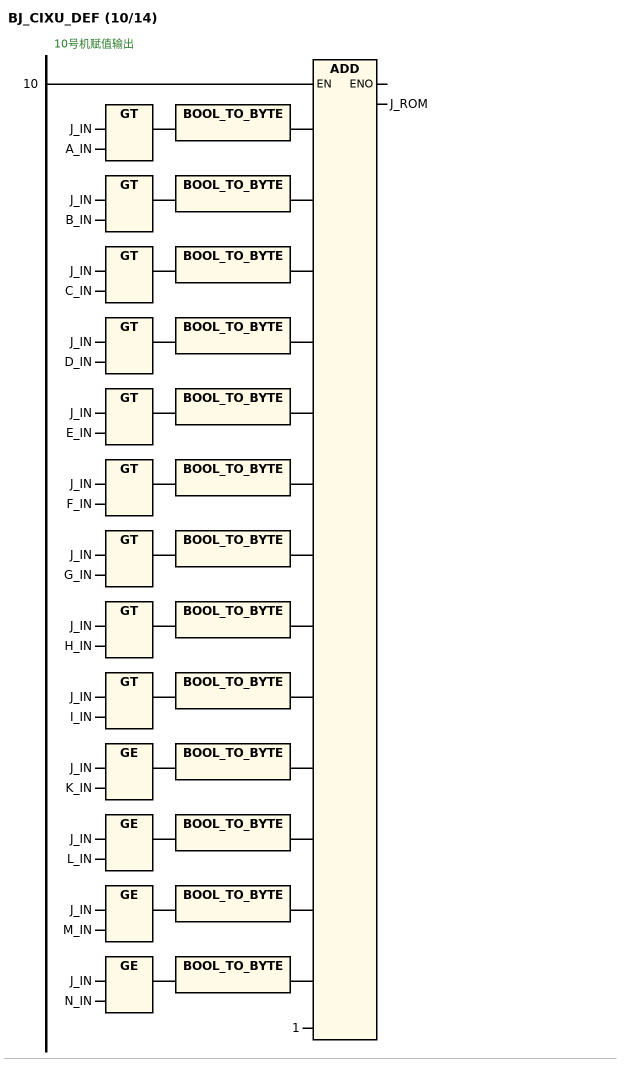
[picture p96: BJ_CIXU_DEF (LD)]
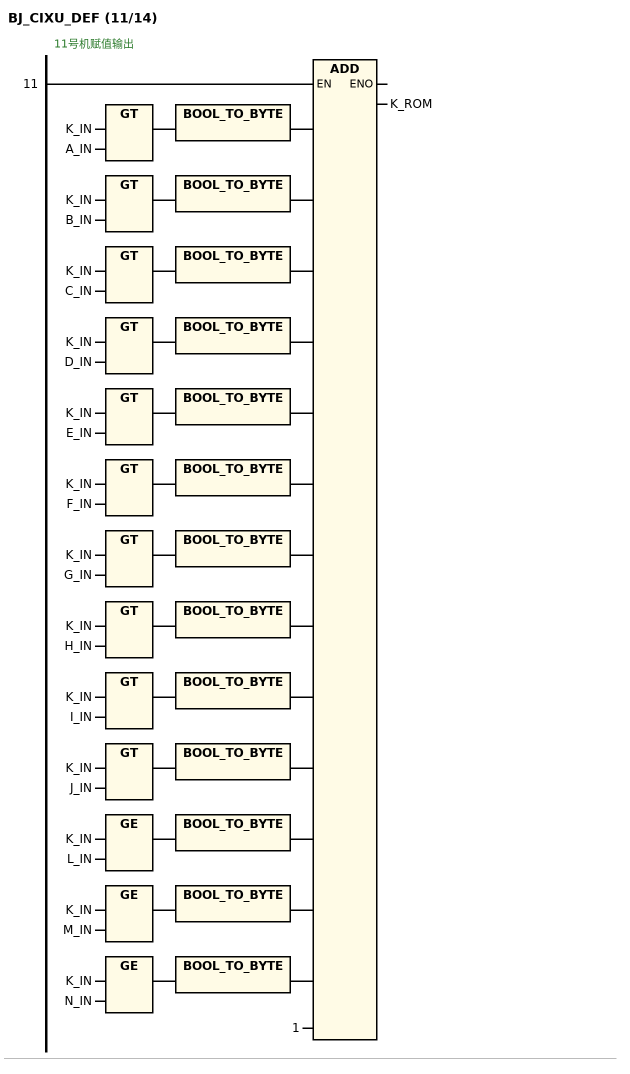
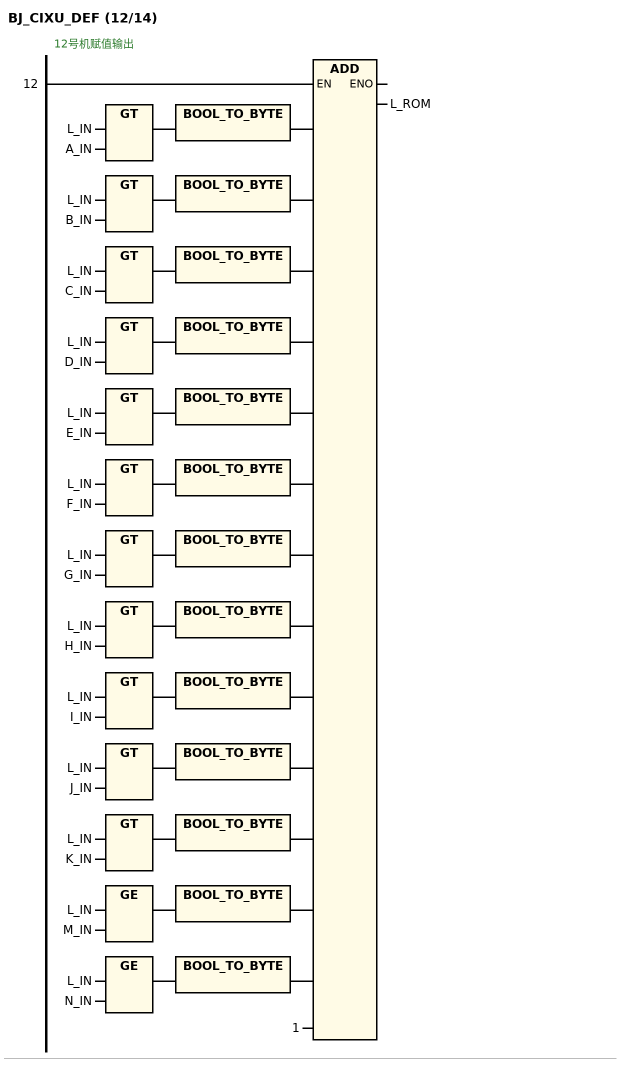
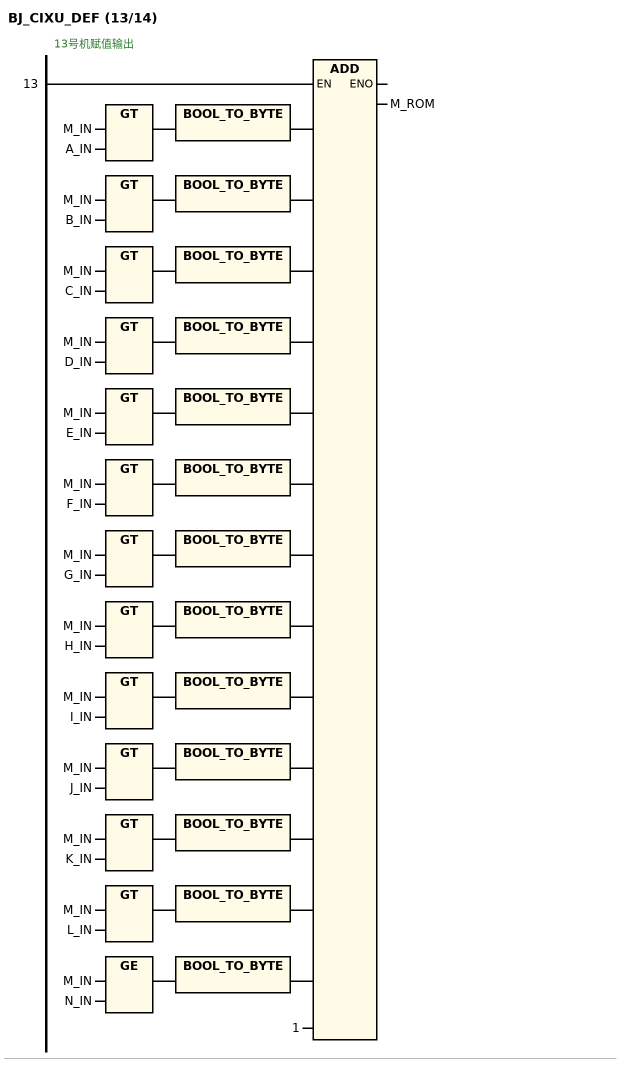
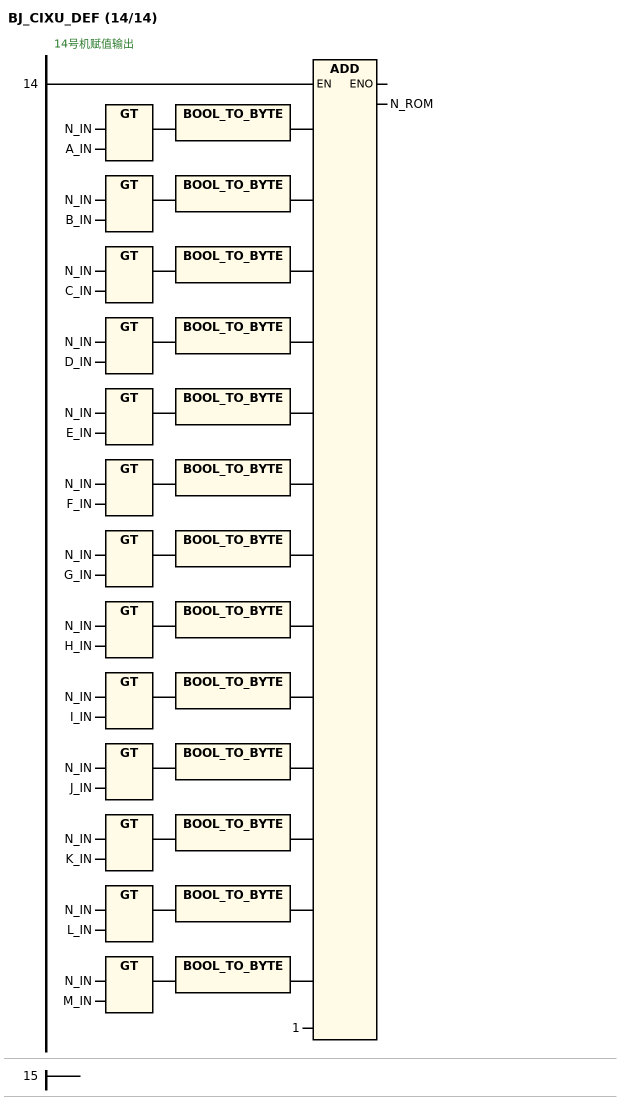
_LD_ (* Ladder Diagram *)
NETWORK 1 (* 1号机赋值输出 *)
	*
		EN --- ADD(BOOL_TO_BYTE(GE(A_IN, B_IN)), BOOL_TO_BYTE(GE(A_IN, C_IN)), BOOL_TO_BYTE(GE(A_IN, D_IN)), BOOL_TO_BYTE(GE(A_IN, E_IN)), BOOL_TO_BYTE(GE(A_IN, F_IN)), BOOL_TO_BYTE(GE(A_IN, G_IN)), BOOL_TO_BYTE(GE(A_IN, H_IN)), BOOL_TO_BYTE(GE(A_IN, I_IN)), BOOL_TO_BYTE(GE(A_IN, J_IN)), BOOL_TO_BYTE(GE(A_IN, K_IN)), BOOL_TO_BYTE(GE(A_IN, L_IN)), BOOL_TO_BYTE(GE(A_IN, M_IN)), BOOL_TO_BYTE(GE(A_IN, N_IN)), 1) => A_ROM
NETWORK 2 (* 2号机赋值输出 *)
	*
		EN --- ADD(BOOL_TO_BYTE(GT(B_IN, A_IN)), BOOL_TO_BYTE(GE(B_IN, C_IN)), BOOL_TO_BYTE(GE(B_IN, D_IN)), BOOL_TO_BYTE(GE(B_IN, E_IN)), BOOL_TO_BYTE(GE(B_IN, F_IN)), BOOL_TO_BYTE(GE(B_IN, G_IN)), BOOL_TO_BYTE(GE(B_IN, H_IN)), BOOL_TO_BYTE(GE(B_IN, I_IN)), BOOL_TO_BYTE(GE(B_IN, J_IN)), BOOL_TO_BYTE(GE(B_IN, K_IN)), BOOL_TO_BYTE(GE(B_IN, L_IN)), BOOL_TO_BYTE(GE(B_IN, M_IN)), BOOL_TO_BYTE(GE(B_IN, N_IN)), 1) => B_ROM
NETWORK 3 (* 3号机赋值输出 *)
	*
		EN --- ADD(BOOL_TO_BYTE(GT(C_IN, A_IN)), BOOL_TO_BYTE(GT(C_IN, B_IN)), BOOL_TO_BYTE(GE(C_IN, D_IN)), BOOL_TO_BYTE(GE(C_IN, E_IN)), BOOL_TO_BYTE(GE(C_IN, F_IN)), BOOL_TO_BYTE(GE(C_IN, G_IN)), BOOL_TO_BYTE(GE(C_IN, H_IN)), BOOL_TO_BYTE(GE(C_IN, I_IN)), BOOL_TO_BYTE(GE(C_IN, J_IN)), BOOL_TO_BYTE(GE(C_IN, K_IN)), BOOL_TO_BYTE(GE(C_IN, L_IN)), BOOL_TO_BYTE(GE(C_IN, M_IN)), BOOL_TO_BYTE(GE(C_IN, N_IN)), 1) => C_ROM
NETWORK 4 (* 4号机赋值输出 *)
	*
		EN --- ADD(BOOL_TO_BYTE(GT(D_IN, A_IN)), BOOL_TO_BYTE(GT(D_IN, B_IN)), BOOL_TO_BYTE(GT(D_IN, C_IN)), BOOL_TO_BYTE(GE(D_IN, E_IN)), BOOL_TO_BYTE(GE(D_IN, F_IN)), BOOL_TO_BYTE(GE(D_IN, G_IN)), BOOL_TO_BYTE(GE(D_IN, H_IN)), BOOL_TO_BYTE(GE(D_IN, I_IN)), BOOL_TO_BYTE(GE(D_IN, J_IN)), BOOL_TO_BYTE(GE(D_IN, K_IN)), BOOL_TO_BYTE(GE(D_IN, L_IN)), BOOL_TO_BYTE(GE(D_IN, M_IN)), BOOL_TO_BYTE(GE(D_IN, N_IN)), 1) => D_ROM
NETWORK 5 (* 5号机赋值输出 *)
	*
		EN --- ADD(BOOL_TO_BYTE(GT(E_IN, A_IN)), BOOL_TO_BYTE(GT(E_IN, B_IN)), BOOL_TO_BYTE(GT(E_IN, C_IN)), BOOL_TO_BYTE(GT(E_IN, D_IN)), BOOL_TO_BYTE(GE(E_IN, F_IN)), BOOL_TO_BYTE(GE(E_IN, G_IN)), BOOL_TO_BYTE(GE(E_IN, H_IN)), BOOL_TO_BYTE(GE(E_IN, I_IN)), BOOL_TO_BYTE(GE(E_IN, J_IN)), BOOL_TO_BYTE(GE(E_IN, K_IN)), BOOL_TO_BYTE(GE(E_IN, L_IN)), BOOL_TO_BYTE(GE(E_IN, M_IN)), BOOL_TO_BYTE(GE(E_IN, N_IN)), 1) => E_ROM
NETWORK 6 (* 6号机赋值输出 *)
	*
		EN --- ADD(BOOL_TO_BYTE(GT(F_IN, A_IN)), BOOL_TO_BYTE(GT(F_IN, B_IN)), BOOL_TO_BYTE(GT(F_IN, C_IN)), BOOL_TO_BYTE(GT(F_IN, D_IN)), BOOL_TO_BYTE(GT(F_IN, E_IN)), BOOL_TO_BYTE(GE(F_IN, G_IN)), BOOL_TO_BYTE(GE(F_IN, H_IN)), BOOL_TO_BYTE(GE(F_IN, I_IN)), BOOL_TO_BYTE(GE(F_IN, J_IN)), BOOL_TO_BYTE(GE(F_IN, K_IN)), BOOL_TO_BYTE(GE(F_IN, L_IN)), BOOL_TO_BYTE(GE(F_IN, M_IN)), BOOL_TO_BYTE(GE(F_IN, N_IN)), 1) => F_ROM
NETWORK 7 (* 7号机赋值输出 *)
	*
		EN --- ADD(BOOL_TO_BYTE(GT(G_IN, A_IN)), BOOL_TO_BYTE(GT(G_IN, B_IN)), BOOL_TO_BYTE(GT(G_IN, C_IN)), BOOL_TO_BYTE(GT(G_IN, D_IN)), BOOL_TO_BYTE(GT(G_IN, E_IN)), BOOL_TO_BYTE(GT(G_IN, F_IN)), BOOL_TO_BYTE(GE(G_IN, H_IN)), BOOL_TO_BYTE(GE(G_IN, I_IN)), BOOL_TO_BYTE(GE(G_IN, J_IN)), BOOL_TO_BYTE(GE(G_IN, K_IN)), BOOL_TO_BYTE(GE(G_IN, L_IN)), BOOL_TO_BYTE(GE(G_IN, M_IN)), BOOL_TO_BYTE(GE(G_IN, N_IN)), 1) => G_ROM
NETWORK 8 (* 8号机赋值输出 *)
	*
		EN --- ADD(BOOL_TO_BYTE(GT(H_IN, A_IN)), BOOL_TO_BYTE(GT(H_IN, B_IN)), BOOL_TO_BYTE(GT(H_IN, C_IN)), BOOL_TO_BYTE(GT(H_IN, D_IN)), BOOL_TO_BYTE(GT(H_IN, E_IN)), BOOL_TO_BYTE(GT(H_IN, F_IN)), BOOL_TO_BYTE(GT(H_IN, G_IN)), BOOL_TO_BYTE(GE(H_IN, I_IN)), BOOL_TO_BYTE(GE(H_IN, J_IN)), BOOL_TO_BYTE(GE(H_IN, K_IN)), BOOL_TO_BYTE(GE(H_IN, L_IN)), BOOL_TO_BYTE(GE(H_IN, M_IN)), BOOL_TO_BYTE(GE(H_IN, N_IN)), 1) => H_ROM
NETWORK 9 (* 9号机赋值输出 *)
	*
		EN --- ADD(BOOL_TO_BYTE(GT(I_IN, A_IN)), BOOL_TO_BYTE(GT(I_IN, B_IN)), BOOL_TO_BYTE(GT(I_IN, C_IN)), BOOL_TO_BYTE(GT(I_IN, D_IN)), BOOL_TO_BYTE(GT(I_IN, E_IN)), BOOL_TO_BYTE(GT(I_IN, F_IN)), BOOL_TO_BYTE(GT(I_IN, G_IN)), BOOL_TO_BYTE(GT(I_IN, H_IN)), BOOL_TO_BYTE(GE(I_IN, J_IN)), BOOL_TO_BYTE(GE(I_IN, K_IN)), BOOL_TO_BYTE(GE(I_IN, L_IN)), BOOL_TO_BYTE(GE(I_IN, M_IN)), BOOL_TO_BYTE(GE(I_IN, N_IN)), 1) => I_ROM
NETWORK 10 (* 10号机赋值输出 *)
	*
		EN --- ADD(BOOL_TO_BYTE(GT(J_IN, A_IN)), BOOL_TO_BYTE(GT(J_IN, B_IN)), BOOL_TO_BYTE(GT(J_IN, C_IN)), BOOL_TO_BYTE(GT(J_IN, D_IN)), BOOL_TO_BYTE(GT(J_IN, E_IN)), BOOL_TO_BYTE(GT(J_IN, F_IN)), BOOL_TO_BYTE(GT(J_IN, G_IN)), BOOL_TO_BYTE(GT(J_IN, H_IN)), BOOL_TO_BYTE(GT(J_IN, I_IN)), BOOL_TO_BYTE(GE(J_IN, K_IN)), BOOL_TO_BYTE(GE(J_IN, L_IN)), BOOL_TO_BYTE(GE(J_IN, M_IN)), BOOL_TO_BYTE(GE(J_IN, N_IN)), 1) => J_ROM
NETWORK 11 (* 11号机赋值输出 *)
	*
		EN --- ADD(BOOL_TO_BYTE(GT(K_IN, A_IN)), BOOL_TO_BYTE(GT(K_IN, B_IN)), BOOL_TO_BYTE(GT(K_IN, C_IN)), BOOL_TO_BYTE(GT(K_IN, D_IN)), BOOL_TO_BYTE(GT(K_IN, E_IN)), BOOL_TO_BYTE(GT(K_IN, F_IN)), BOOL_TO_BYTE(GT(K_IN, G_IN)), BOOL_TO_BYTE(GT(K_IN, H_IN)), BOOL_TO_BYTE(GT(K_IN, I_IN)), BOOL_TO_BYTE(GT(K_IN, J_IN)), BOOL_TO_BYTE(GE(K_IN, L_IN)), BOOL_TO_BYTE(GE(K_IN, M_IN)), BOOL_TO_BYTE(GE(K_IN, N_IN)), 1) => K_ROM
NETWORK 12 (* 12号机赋值输出 *)
	*
		EN --- ADD(BOOL_TO_BYTE(GT(L_IN, A_IN)), BOOL_TO_BYTE(GT(L_IN, B_IN)), BOOL_TO_BYTE(GT(L_IN, C_IN)), BOOL_TO_BYTE(GT(L_IN, D_IN)), BOOL_TO_BYTE(GT(L_IN, E_IN)), BOOL_TO_BYTE(GT(L_IN, F_IN)), BOOL_TO_BYTE(GT(L_IN, G_IN)), BOOL_TO_BYTE(GT(L_IN, H_IN)), BOOL_TO_BYTE(GT(L_IN, I_IN)), BOOL_TO_BYTE(GT(L_IN, J_IN)), BOOL_TO_BYTE(GT(L_IN, K_IN)), BOOL_TO_BYTE(GE(L_IN, M_IN)), BOOL_TO_BYTE(GE(L_IN, N_IN)), 1) => L_ROM
NETWORK 13 (* 13号机赋值输出 *)
	*
		EN --- ADD(BOOL_TO_BYTE(GT(M_IN, A_IN)), BOOL_TO_BYTE(GT(M_IN, B_IN)), BOOL_TO_BYTE(GT(M_IN, C_IN)), BOOL_TO_BYTE(GT(M_IN, D_IN)), BOOL_TO_BYTE(GT(M_IN, E_IN)), BOOL_TO_BYTE(GT(M_IN, F_IN)), BOOL_TO_BYTE(GT(M_IN, G_IN)), BOOL_TO_BYTE(GT(M_IN, H_IN)), BOOL_TO_BYTE(GT(M_IN, I_IN)), BOOL_TO_BYTE(GT(M_IN, J_IN)), BOOL_TO_BYTE(GT(M_IN, K_IN)), BOOL_TO_BYTE(GT(M_IN, L_IN)), BOOL_TO_BYTE(GE(M_IN, N_IN)), 1) => M_ROM
NETWORK 14 (* 14号机赋值输出 *)
	*
		EN --- ADD(BOOL_TO_BYTE(GT(N_IN, A_IN)), BOOL_TO_BYTE(GT(N_IN, B_IN)), BOOL_TO_BYTE(GT(N_IN, C_IN)), BOOL_TO_BYTE(GT(N_IN, D_IN)), BOOL_TO_BYTE(GT(N_IN, E_IN)), BOOL_TO_BYTE(GT(N_IN, F_IN)), BOOL_TO_BYTE(GT(N_IN, G_IN)), BOOL_TO_BYTE(GT(N_IN, H_IN)), BOOL_TO_BYTE(GT(N_IN, I_IN)), BOOL_TO_BYTE(GT(N_IN, J_IN)), BOOL_TO_BYTE(GT(N_IN, K_IN)), BOOL_TO_BYTE(GT(N_IN, L_IN)), BOOL_TO_BYTE(GT(N_IN, M_IN)), 1) => N_ROM
NETWORK 15
	*
_END_LD_
(* the same logic as Structured Text *)
(* Network 1: 1号机赋值输出 *)
A_ROM := BOOL_TO_BYTE(A_IN >= B_IN) + BOOL_TO_BYTE(A_IN >= C_IN) + BOOL_TO_BYTE(A_IN >= D_IN) + BOOL_TO_BYTE(A_IN >= E_IN) + BOOL_TO_BYTE(A_IN >= F_IN) + BOOL_TO_BYTE(A_IN >= G_IN) + BOOL_TO_BYTE(A_IN >= H_IN) + BOOL_TO_BYTE(A_IN >= I_IN) + BOOL_TO_BYTE(A_IN >= J_IN) + BOOL_TO_BYTE(A_IN >= K_IN) + BOOL_TO_BYTE(A_IN >= L_IN) + BOOL_TO_BYTE(A_IN >= M_IN) + BOOL_TO_BYTE(A_IN >= N_IN) + 1;
(* Network 2: 2号机赋值输出 *)
B_ROM := BOOL_TO_BYTE(B_IN > A_IN) + BOOL_TO_BYTE(B_IN >= C_IN) + BOOL_TO_BYTE(B_IN >= D_IN) + BOOL_TO_BYTE(B_IN >= E_IN) + BOOL_TO_BYTE(B_IN >= F_IN) + BOOL_TO_BYTE(B_IN >= G_IN) + BOOL_TO_BYTE(B_IN >= H_IN) + BOOL_TO_BYTE(B_IN >= I_IN) + BOOL_TO_BYTE(B_IN >= J_IN) + BOOL_TO_BYTE(B_IN >= K_IN) + BOOL_TO_BYTE(B_IN >= L_IN) + BOOL_TO_BYTE(B_IN >= M_IN) + BOOL_TO_BYTE(B_IN >= N_IN) + 1;
(* Network 3: 3号机赋值输出 *)
C_ROM := BOOL_TO_BYTE(C_IN > A_IN) + BOOL_TO_BYTE(C_IN > B_IN) + BOOL_TO_BYTE(C_IN >= D_IN) + BOOL_TO_BYTE(C_IN >= E_IN) + BOOL_TO_BYTE(C_IN >= F_IN) + BOOL_TO_BYTE(C_IN >= G_IN) + BOOL_TO_BYTE(C_IN >= H_IN) + BOOL_TO_BYTE(C_IN >= I_IN) + BOOL_TO_BYTE(C_IN >= J_IN) + BOOL_TO_BYTE(C_IN >= K_IN) + BOOL_TO_BYTE(C_IN >= L_IN) + BOOL_TO_BYTE(C_IN >= M_IN) + BOOL_TO_BYTE(C_IN >= N_IN) + 1;
(* Network 4: 4号机赋值输出 *)
D_ROM := BOOL_TO_BYTE(D_IN > A_IN) + BOOL_TO_BYTE(D_IN > B_IN) + BOOL_TO_BYTE(D_IN > C_IN) + BOOL_TO_BYTE(D_IN >= E_IN) + BOOL_TO_BYTE(D_IN >= F_IN) + BOOL_TO_BYTE(D_IN >= G_IN) + BOOL_TO_BYTE(D_IN >= H_IN) + BOOL_TO_BYTE(D_IN >= I_IN) + BOOL_TO_BYTE(D_IN >= J_IN) + BOOL_TO_BYTE(D_IN >= K_IN) + BOOL_TO_BYTE(D_IN >= L_IN) + BOOL_TO_BYTE(D_IN >= M_IN) + BOOL_TO_BYTE(D_IN >= N_IN) + 1;
(* Network 5: 5号机赋值输出 *)
E_ROM := BOOL_TO_BYTE(E_IN > A_IN) + BOOL_TO_BYTE(E_IN > B_IN) + BOOL_TO_BYTE(E_IN > C_IN) + BOOL_TO_BYTE(E_IN > D_IN) + BOOL_TO_BYTE(E_IN >= F_IN) + BOOL_TO_BYTE(E_IN >= G_IN) + BOOL_TO_BYTE(E_IN >= H_IN) + BOOL_TO_BYTE(E_IN >= I_IN) + BOOL_TO_BYTE(E_IN >= J_IN) + BOOL_TO_BYTE(E_IN >= K_IN) + BOOL_TO_BYTE(E_IN >= L_IN) + BOOL_TO_BYTE(E_IN >= M_IN) + BOOL_TO_BYTE(E_IN >= N_IN) + 1;
(* Network 6: 6号机赋值输出 *)
F_ROM := BOOL_TO_BYTE(F_IN > A_IN) + BOOL_TO_BYTE(F_IN > B_IN) + BOOL_TO_BYTE(F_IN > C_IN) + BOOL_TO_BYTE(F_IN > D_IN) + BOOL_TO_BYTE(F_IN > E_IN) + BOOL_TO_BYTE(F_IN >= G_IN) + BOOL_TO_BYTE(F_IN >= H_IN) + BOOL_TO_BYTE(F_IN >= I_IN) + BOOL_TO_BYTE(F_IN >= J_IN) + BOOL_TO_BYTE(F_IN >= K_IN) + BOOL_TO_BYTE(F_IN >= L_IN) + BOOL_TO_BYTE(F_IN >= M_IN) + BOOL_TO_BYTE(F_IN >= N_IN) + 1;
(* Network 7: 7号机赋值输出 *)
G_ROM := BOOL_TO_BYTE(G_IN > A_IN) + BOOL_TO_BYTE(G_IN > B_IN) + BOOL_TO_BYTE(G_IN > C_IN) + BOOL_TO_BYTE(G_IN > D_IN) + BOOL_TO_BYTE(G_IN > E_IN) + BOOL_TO_BYTE(G_IN > F_IN) + BOOL_TO_BYTE(G_IN >= H_IN) + BOOL_TO_BYTE(G_IN >= I_IN) + BOOL_TO_BYTE(G_IN >= J_IN) + BOOL_TO_BYTE(G_IN >= K_IN) + BOOL_TO_BYTE(G_IN >= L_IN) + BOOL_TO_BYTE(G_IN >= M_IN) + BOOL_TO_BYTE(G_IN >= N_IN) + 1;
(* Network 8: 8号机赋值输出 *)
H_ROM := BOOL_TO_BYTE(H_IN > A_IN) + BOOL_TO_BYTE(H_IN > B_IN) + BOOL_TO_BYTE(H_IN > C_IN) + BOOL_TO_BYTE(H_IN > D_IN) + BOOL_TO_BYTE(H_IN > E_IN) + BOOL_TO_BYTE(H_IN > F_IN) + BOOL_TO_BYTE(H_IN > G_IN) + BOOL_TO_BYTE(H_IN >= I_IN) + BOOL_TO_BYTE(H_IN >= J_IN) + BOOL_TO_BYTE(H_IN >= K_IN) + BOOL_TO_BYTE(H_IN >= L_IN) + BOOL_TO_BYTE(H_IN >= M_IN) + BOOL_TO_BYTE(H_IN >= N_IN) + 1;
(* Network 9: 9号机赋值输出 *)
I_ROM := BOOL_TO_BYTE(I_IN > A_IN) + BOOL_TO_BYTE(I_IN > B_IN) + BOOL_TO_BYTE(I_IN > C_IN) + BOOL_TO_BYTE(I_IN > D_IN) + BOOL_TO_BYTE(I_IN > E_IN) + BOOL_TO_BYTE(I_IN > F_IN) + BOOL_TO_BYTE(I_IN > G_IN) + BOOL_TO_BYTE(I_IN > H_IN) + BOOL_TO_BYTE(I_IN >= J_IN) + BOOL_TO_BYTE(I_IN >= K_IN) + BOOL_TO_BYTE(I_IN >= L_IN) + BOOL_TO_BYTE(I_IN >= M_IN) + BOOL_TO_BYTE(I_IN >= N_IN) + 1;
(* Network 10: 10号机赋值输出 *)
J_ROM := BOOL_TO_BYTE(J_IN > A_IN) + BOOL_TO_BYTE(J_IN > B_IN) + BOOL_TO_BYTE(J_IN > C_IN) + BOOL_TO_BYTE(J_IN > D_IN) + BOOL_TO_BYTE(J_IN > E_IN) + BOOL_TO_BYTE(J_IN > F_IN) + BOOL_TO_BYTE(J_IN > G_IN) + BOOL_TO_BYTE(J_IN > H_IN) + BOOL_TO_BYTE(J_IN > I_IN) + BOOL_TO_BYTE(J_IN >= K_IN) + BOOL_TO_BYTE(J_IN >= L_IN) + BOOL_TO_BYTE(J_IN >= M_IN) + BOOL_TO_BYTE(J_IN >= N_IN) + 1;
(* Network 11: 11号机赋值输出 *)
K_ROM := BOOL_TO_BYTE(K_IN > A_IN) + BOOL_TO_BYTE(K_IN > B_IN) + BOOL_TO_BYTE(K_IN > C_IN) + BOOL_TO_BYTE(K_IN > D_IN) + BOOL_TO_BYTE(K_IN > E_IN) + BOOL_TO_BYTE(K_IN > F_IN) + BOOL_TO_BYTE(K_IN > G_IN) + BOOL_TO_BYTE(K_IN > H_IN) + BOOL_TO_BYTE(K_IN > I_IN) + BOOL_TO_BYTE(K_IN > J_IN) + BOOL_TO_BYTE(K_IN >= L_IN) + BOOL_TO_BYTE(K_IN >= M_IN) + BOOL_TO_BYTE(K_IN >= N_IN) + 1;
(* Network 12: 12号机赋值输出 *)
L_ROM := BOOL_TO_BYTE(L_IN > A_IN) + BOOL_TO_BYTE(L_IN > B_IN) + BOOL_TO_BYTE(L_IN > C_IN) + BOOL_TO_BYTE(L_IN > D_IN) + BOOL_TO_BYTE(L_IN > E_IN) + BOOL_TO_BYTE(L_IN > F_IN) + BOOL_TO_BYTE(L_IN > G_IN) + BOOL_TO_BYTE(L_IN > H_IN) + BOOL_TO_BYTE(L_IN > I_IN) + BOOL_TO_BYTE(L_IN > J_IN) + BOOL_TO_BYTE(L_IN > K_IN) + BOOL_TO_BYTE(L_IN >= M_IN) + BOOL_TO_BYTE(L_IN >= N_IN) + 1;
(* Network 13: 13号机赋值输出 *)
M_ROM := BOOL_TO_BYTE(M_IN > A_IN) + BOOL_TO_BYTE(M_IN > B_IN) + BOOL_TO_BYTE(M_IN > C_IN) + BOOL_TO_BYTE(M_IN > D_IN) + BOOL_TO_BYTE(M_IN > E_IN) + BOOL_TO_BYTE(M_IN > F_IN) + BOOL_TO_BYTE(M_IN > G_IN) + BOOL_TO_BYTE(M_IN > H_IN) + BOOL_TO_BYTE(M_IN > I_IN) + BOOL_TO_BYTE(M_IN > J_IN) + BOOL_TO_BYTE(M_IN > K_IN) + BOOL_TO_BYTE(M_IN > L_IN) + BOOL_TO_BYTE(M_IN >= N_IN) + 1;
(* Network 14: 14号机赋值输出 *)
N_ROM := BOOL_TO_BYTE(N_IN > A_IN) + BOOL_TO_BYTE(N_IN > B_IN) + BOOL_TO_BYTE(N_IN > C_IN) + BOOL_TO_BYTE(N_IN > D_IN) + BOOL_TO_BYTE(N_IN > E_IN) + BOOL_TO_BYTE(N_IN > F_IN) + BOOL_TO_BYTE(N_IN > G_IN) + BOOL_TO_BYTE(N_IN > H_IN) + BOOL_TO_BYTE(N_IN > I_IN) + BOOL_TO_BYTE(N_IN > J_IN) + BOOL_TO_BYTE(N_IN > K_IN) + BOOL_TO_BYTE(N_IN > L_IN) + BOOL_TO_BYTE(N_IN > M_IN) + 1;
(* Network 15 *)
END_FUNCTION_BLOCK

(* POU DEF_PAIXU, LD *)
FUNCTION_BLOCK DEF_PAIXU
VAR_INPUT
	A_IN: BOOL;
	A_ROM: BYTE;
	B_IN: BOOL;
	B_ROM: BYTE;
	C_IN: BOOL;
	C_ROM: BYTE;
	D_IN: BOOL;
	D_ROM: BYTE;
	E_IN: BOOL;
	E_ROM: BYTE;
	F_IN: BOOL;
	F_ROM: BYTE;
	G_IN: BOOL;
	G_ROM: BYTE;
	H_IN: BOOL;
	H_ROM: BYTE;
	I_IN: BOOL;
	I_ROM: BYTE;
	J_IN: BOOL;
	J_ROM: BYTE;
	K_IN: BOOL;
	K_ROM: BYTE;
	L_IN: BOOL;
	L_ROM: BYTE;
	M_IN: BOOL;
	M_ROM: BYTE;
	N_IN: BOOL;
	N_ROM: BYTE;
	ROM_SHU: WORD;
	PSH_IN: BOOL;
END_VAR
VAR_OUTPUT
	A_DZ: BOOL;
	B_DZ: BOOL;
	C_DZ: BOOL;
	D_DZ: BOOL;
	E_DZ: BOOL;
	F_DZ: BOOL;
	G_DZ: BOOL;
	H_DZ: BOOL;
	I_DZ: BOOL;
	J_DZ: BOOL;
	K_DZ: BOOL;
	L_DZ: BOOL;
	M_DZ: BOOL;
	N_DZ: BOOL;
	A_KA: BOOL;
	B_KA: BOOL;
	C_KA: BOOL;
	D_KA: BOOL;
	E_KA: BOOL;
	F_KA: BOOL;
	G_KA: BOOL;
	H_KA: BOOL;
	  I_KA: BOOL;
	J_KA: BOOL;
	K_KA: BOOL;
	L_KA: BOOL;
       M_KA: BOOL;
	N_KA: BOOL;
	FJ_ROM: BYTE;
	ROM: BYTE;
END_VAR
VAR
	INPUT_KA: BOOL;
	A_0: BOOL;
	B_0: BOOL;
	C_0: BOOL;
	D_0: BOOL;
	F_0: BOOL;
	E_0: BOOL;
	G_0: BOOL;
	H_0: BOOL;

	A_FJ: BOOL;
	B_FJ: BOOL;
	C_FJ: BOOL;
	D_FJ: BOOL;
	E_FJ: BOOL;
	F_FJ: BOOL;
	G_FJ: BOOL;
	H_FJ: BOOL;
	I_0: BOOL;

	J_FJ: BOOL;
	J_0: BOOL;
	I_FJ: BOOL;
	KA_FJ: BOOL;
	ROM_1: BOOL;
	ROM_2: BOOL;
	ROM_3: BOOL;
	ROM_4: BOOL;
	ROM_10: BOOL;
	ROM_9: BOOL;
	ROM_8: BOOL;
	ROM_7: BOOL;
	ROM_6: BOOL;
	ROM_5: BOOL;
	FJ_CTU: CTU;
	CTU_Q: BOOL;
	CV: WORD;
	CV_0: BOOL;
	CV_1: BOOL;
	CV_2: BOOL;
	CV_3: BOOL;
	CV_4: BOOL;
	CV_5: BOOL;
	CV_6: BOOL;
	CV_7: BOOL;
	CV_8: BOOL;
	CV_9: BOOL;
	KAIKU_SHU: WORD;
	ROM_0: BOOL;
	KU_SHU: WORD;
	ROM_11: BOOL;
	ROM_12: BOOL;
	ROM_13: BOOL;
	ROM_14: BOOL;
	K_0: BOOL;
	K_FJ: BOOL;
	L_0: BOOL;
	L_FJ: BOOL;
	M_0: BOOL;
	M_FJ: BOOL;
	N_0: BOOL;
	N_FJ: BOOL;
	CV_10: BOOL;
	CV_11: BOOL;
	CV_12: BOOL;
	CV_13: BOOL;
	A_15: BOOL;
	B_15: BOOL;
	C_15: BOOL;
	D_15: BOOL;
	E_15: BOOL;
	F_15: BOOL;
	H_15: BOOL;
	I_15: BOOL;
	J_15: BOOL;
	K_15: BOOL;
	L_15: BOOL;
	M_15: BOOL;
	N_15: BOOL;
	G_15: BOOL;
END_VAR
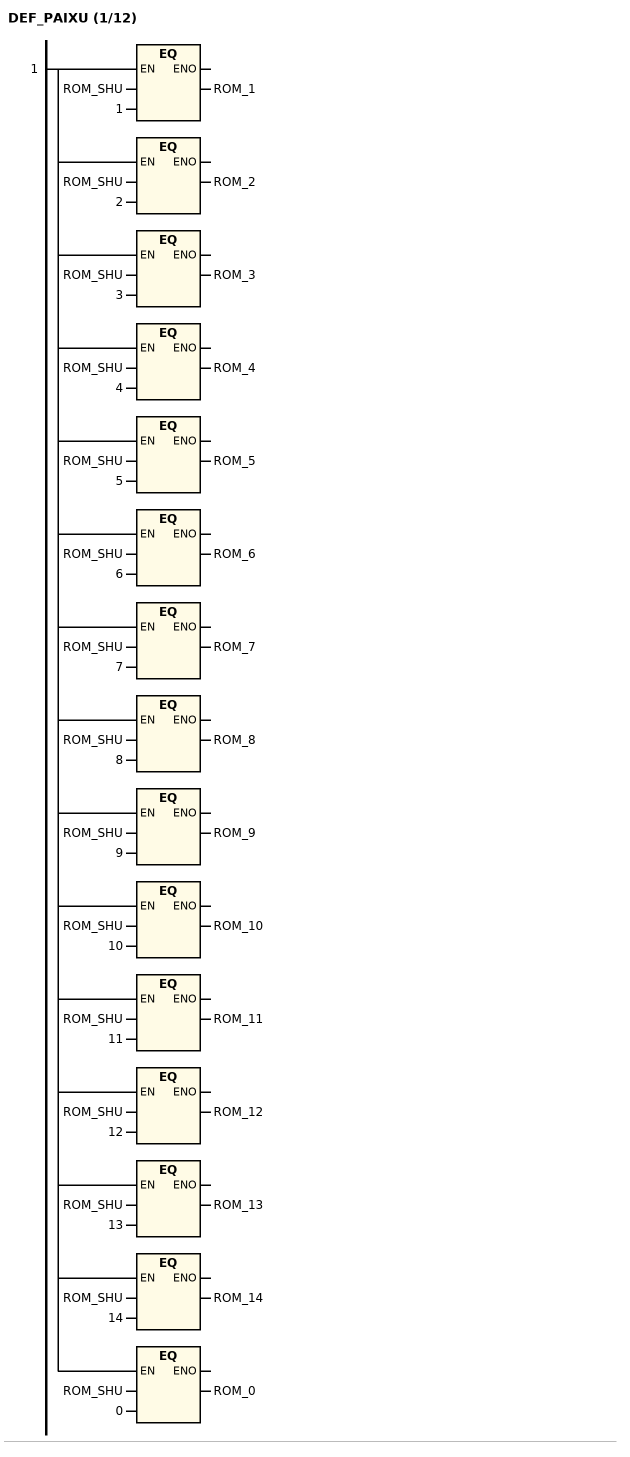
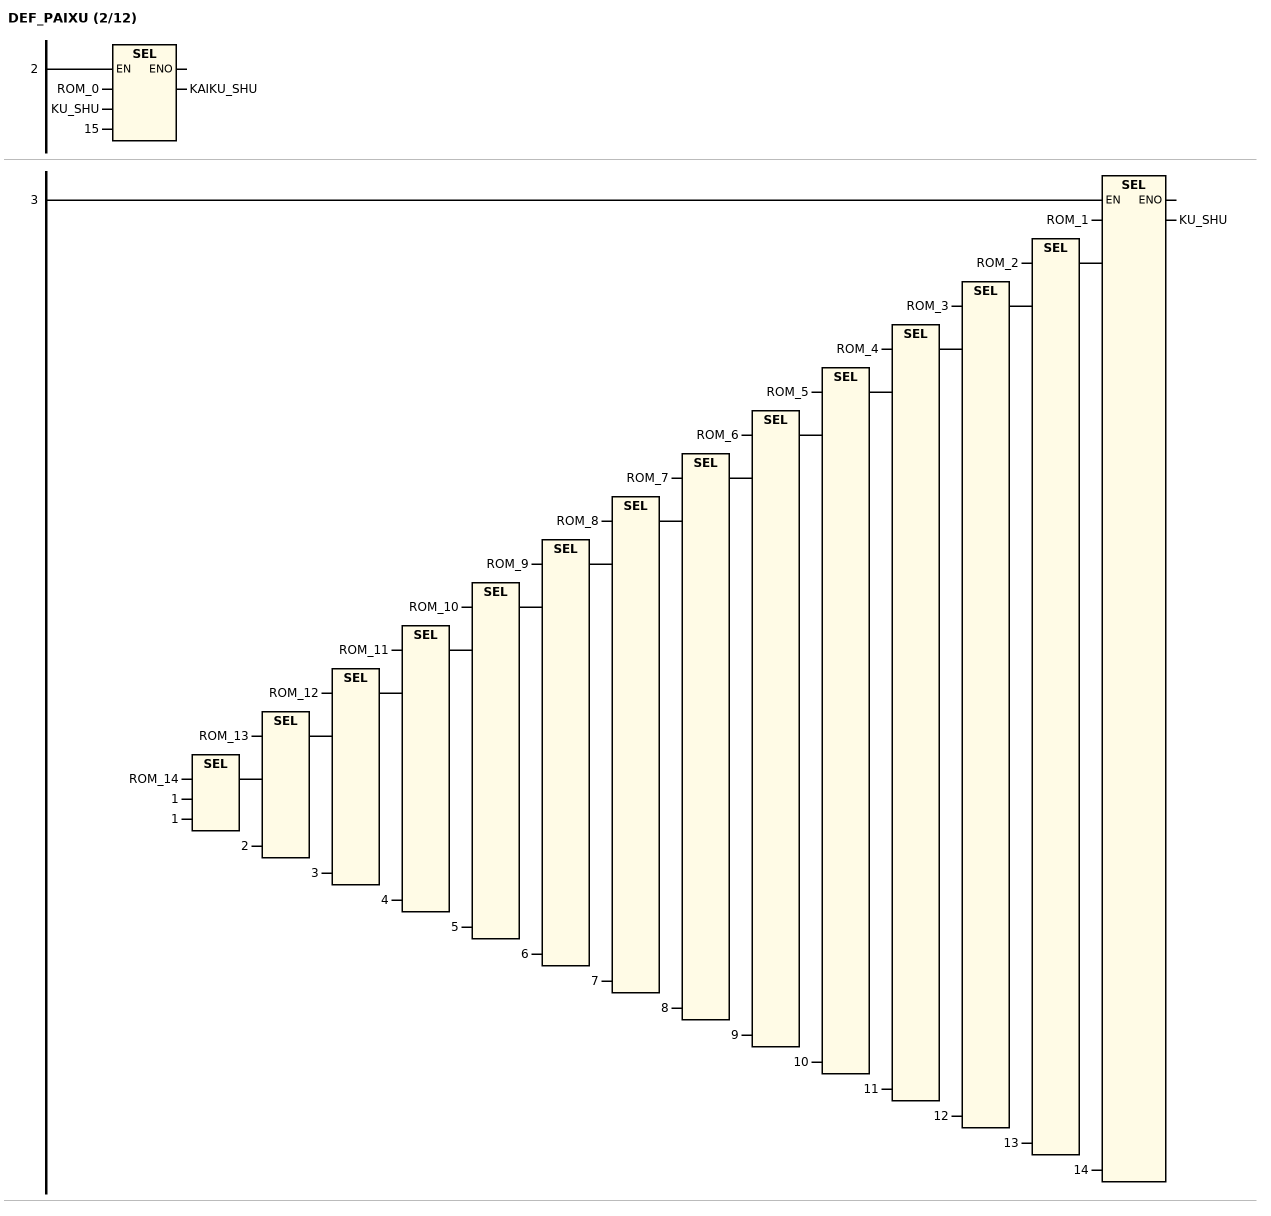
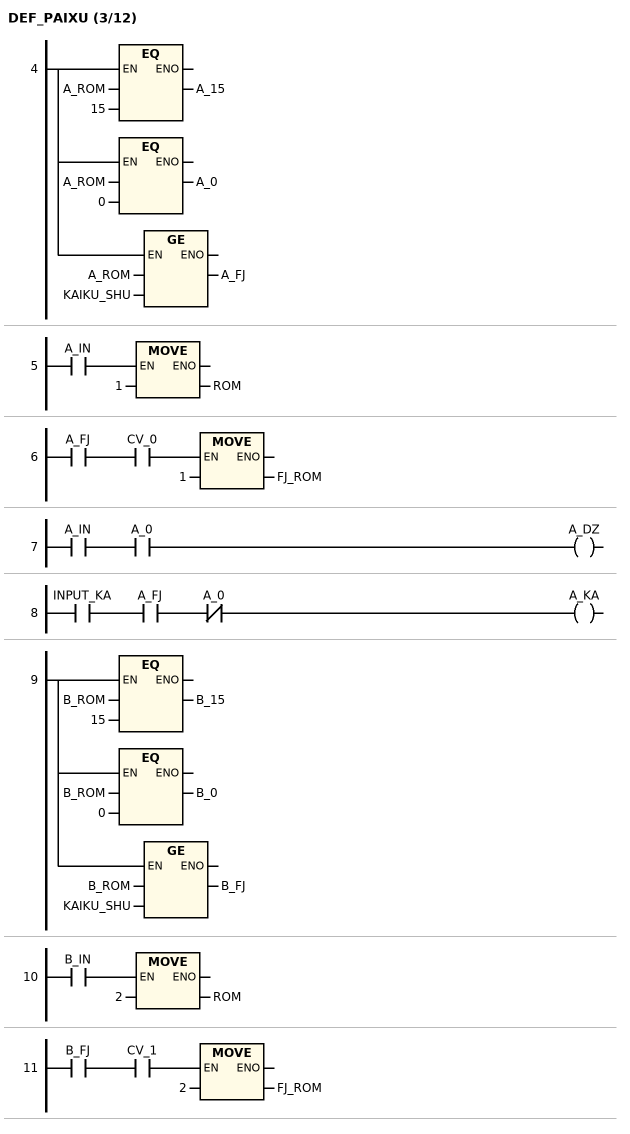
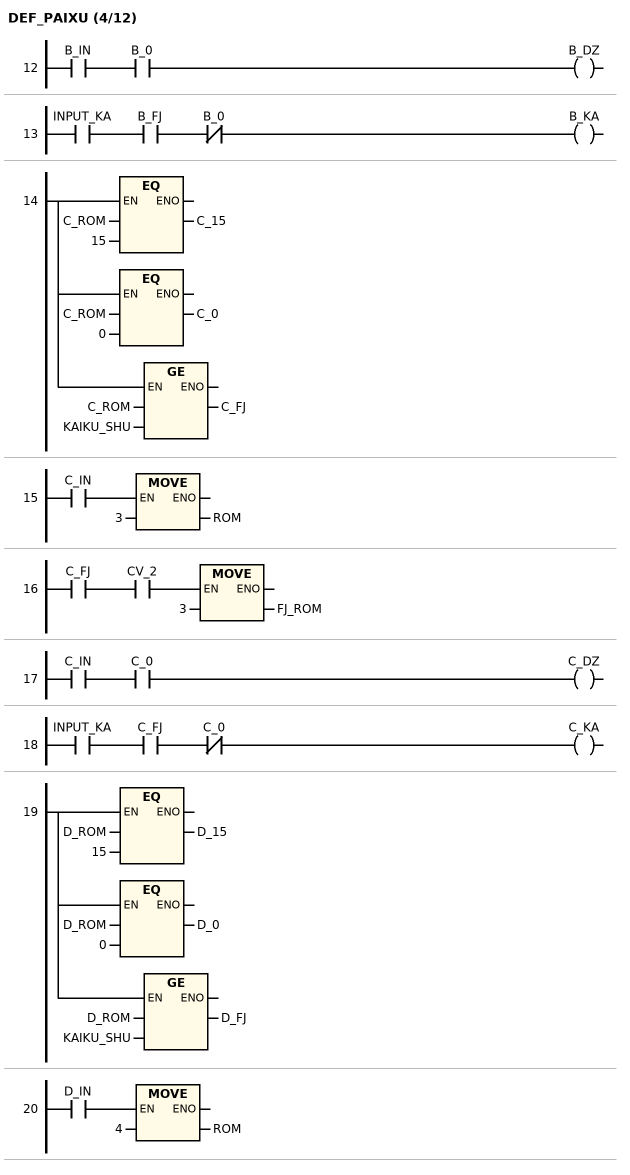
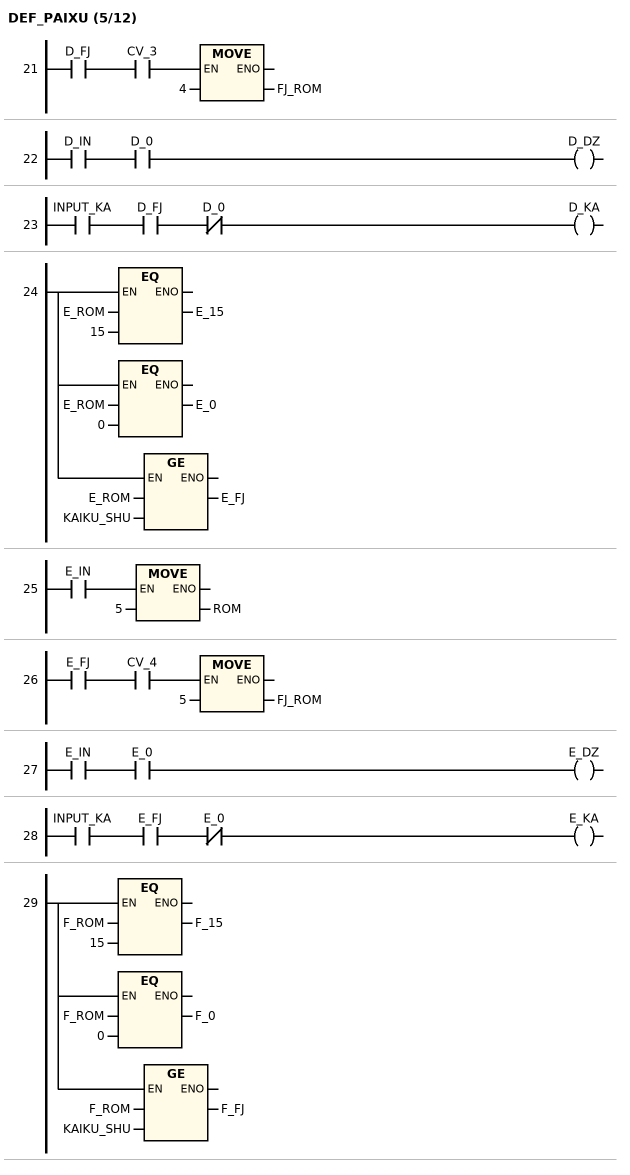
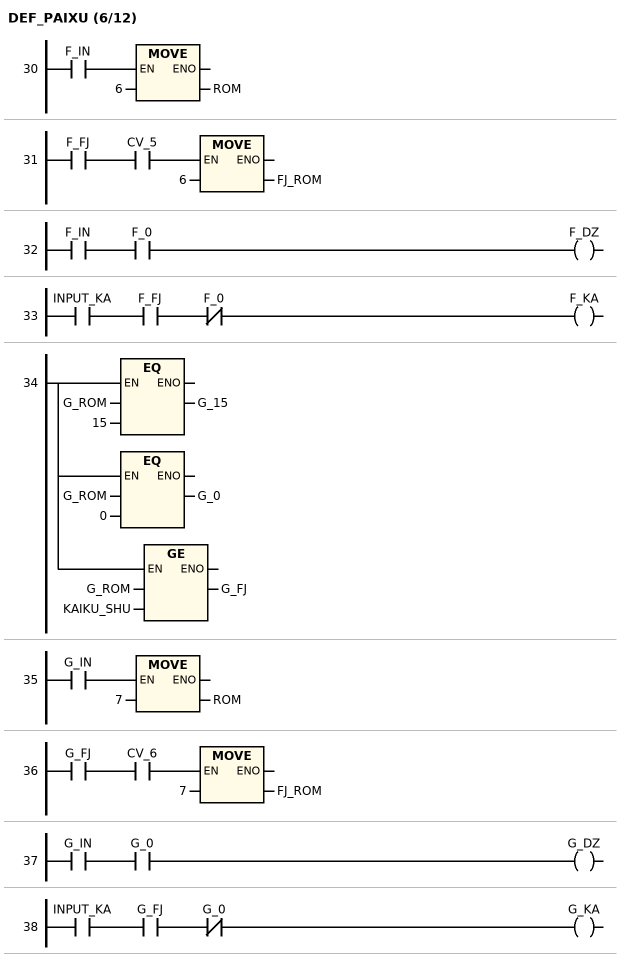
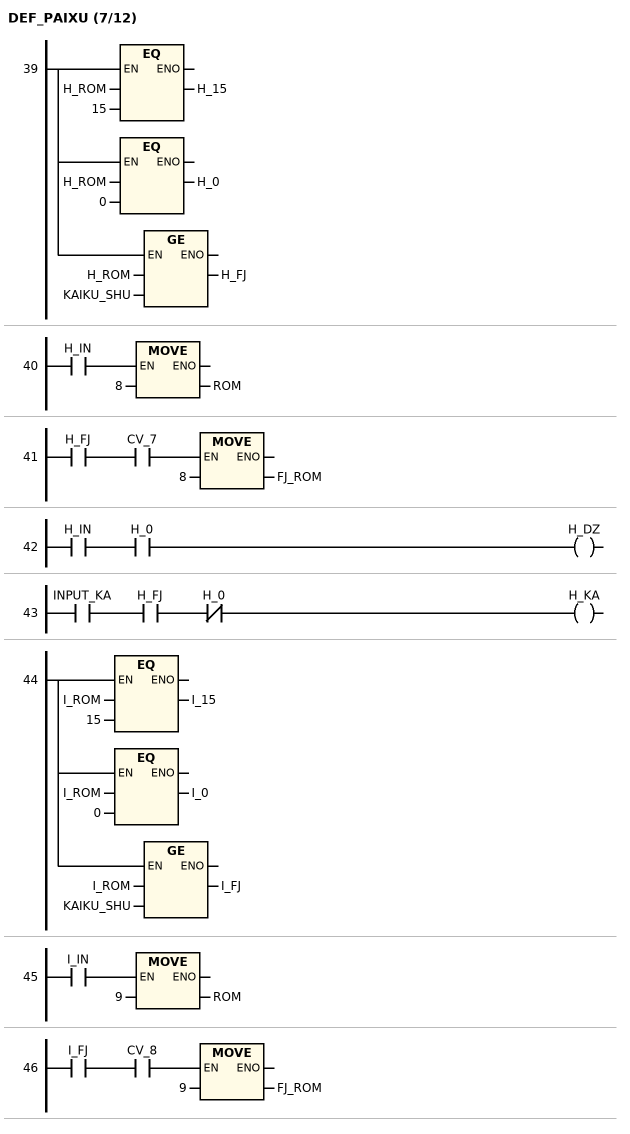
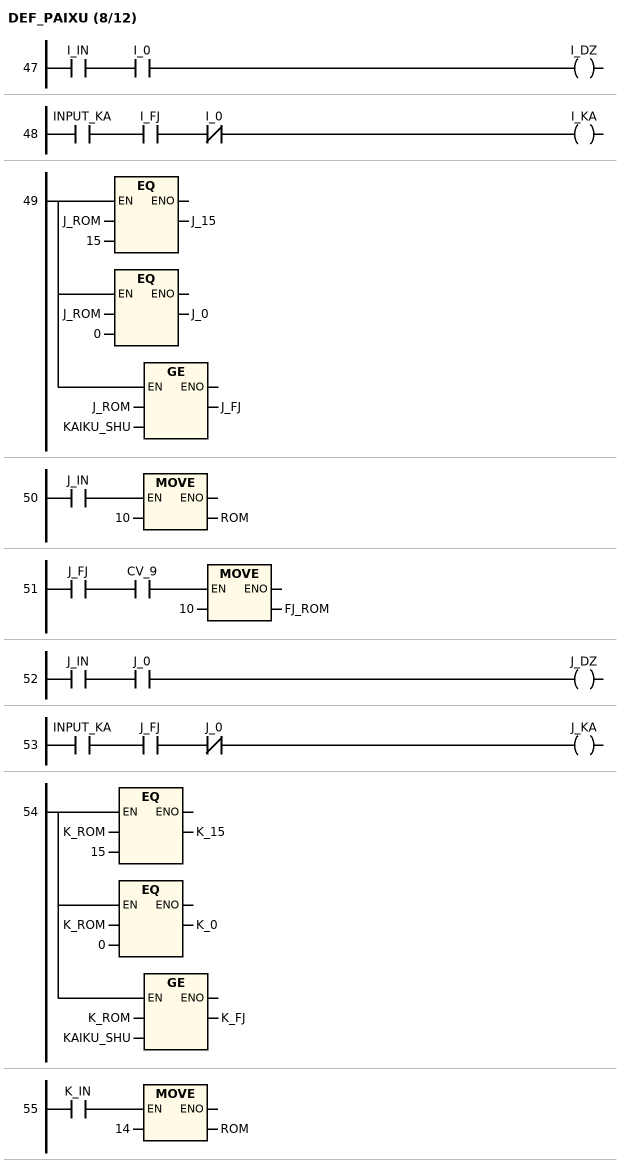
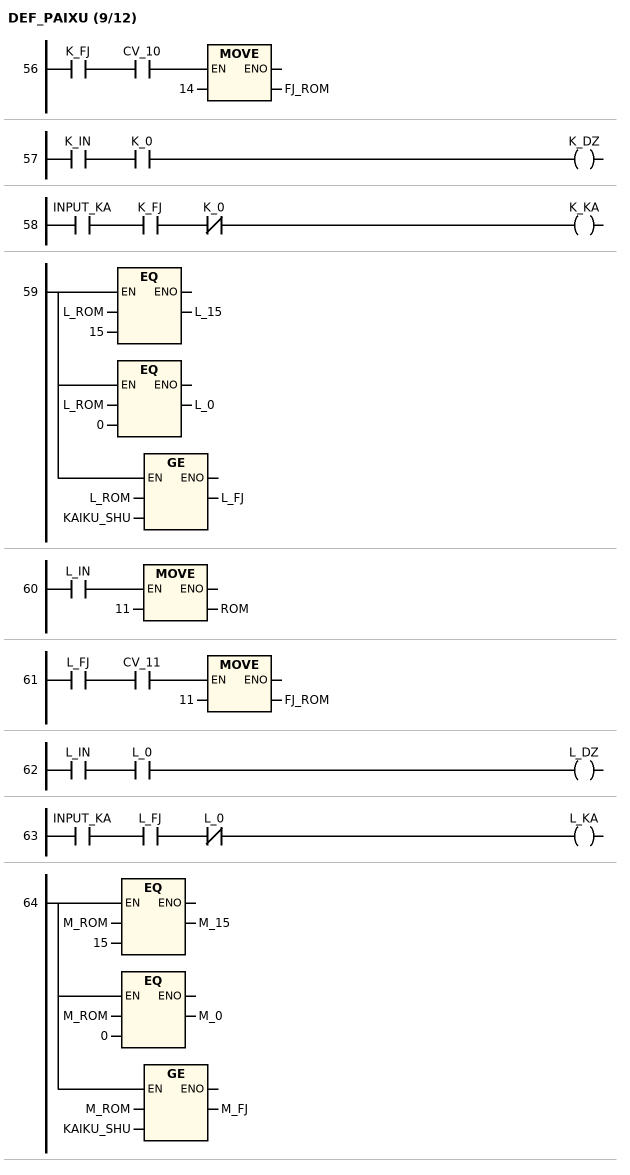
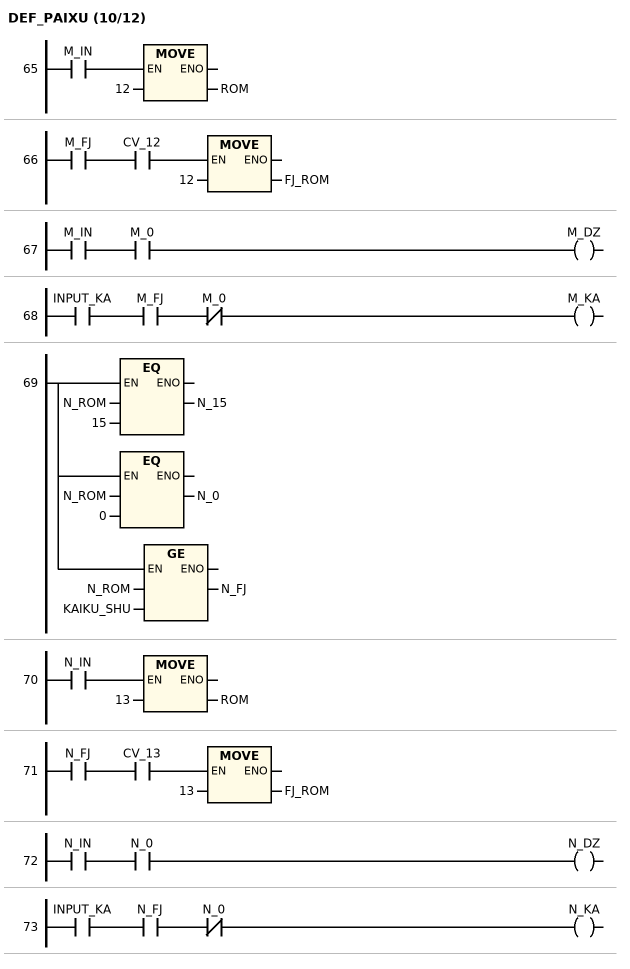
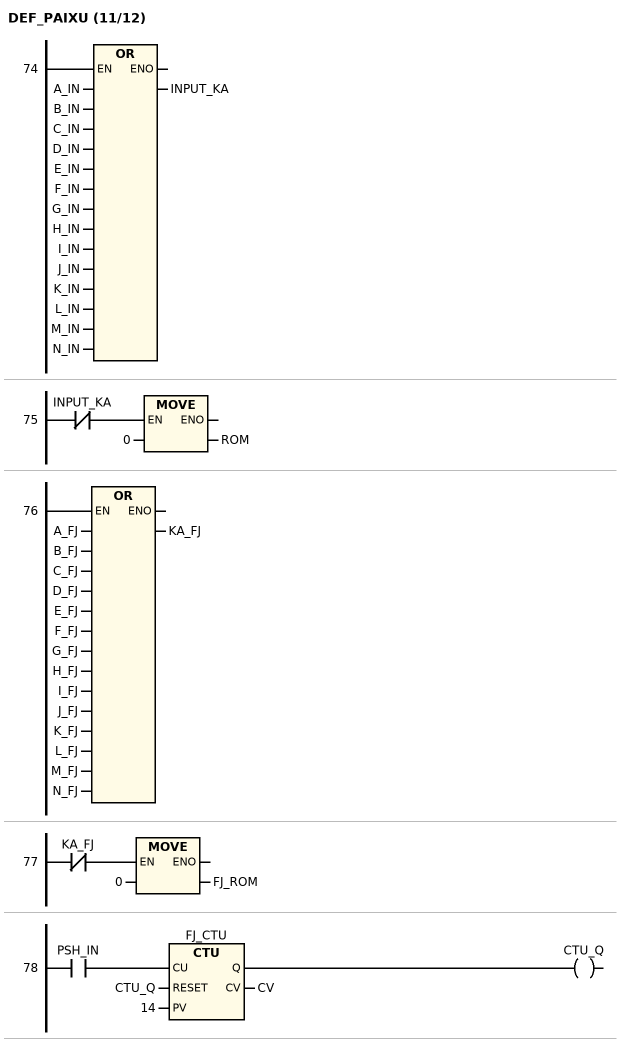
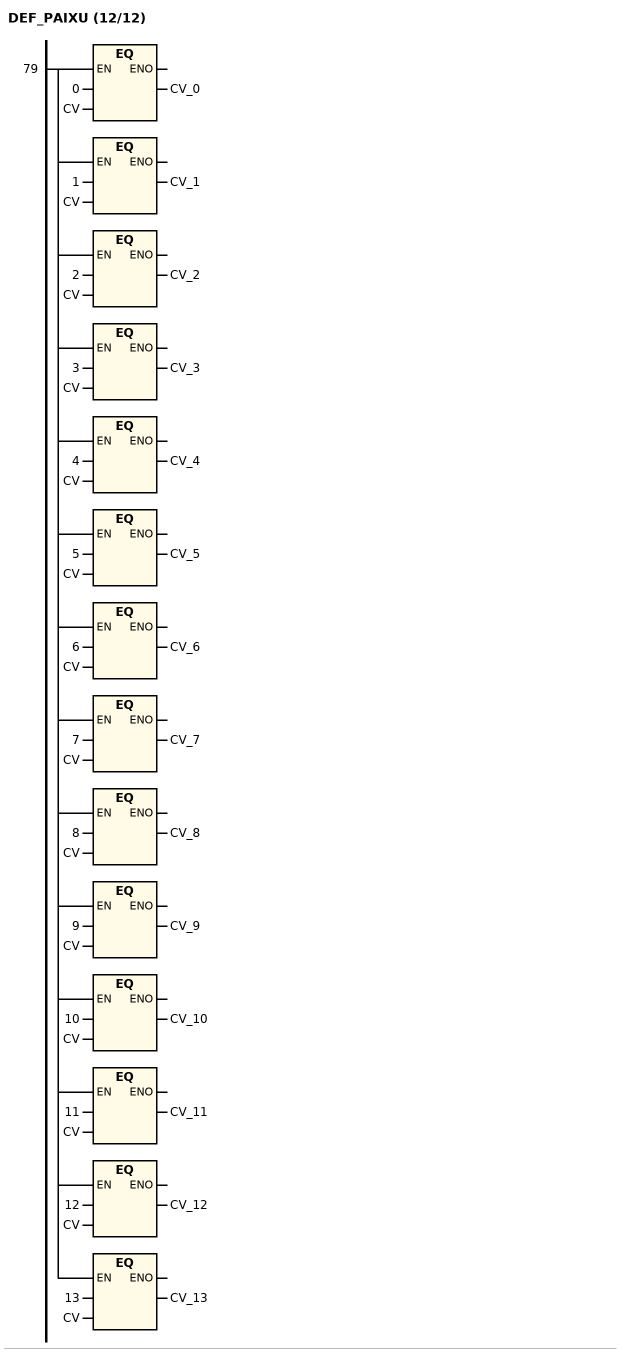
_LD_ (* Ladder Diagram *)
NETWORK 1
	*
		EN --- EQ(ROM_SHU, 1) => ROM_1
		EN --- EQ(ROM_SHU, 2) => ROM_2
		EN --- EQ(ROM_SHU, 3) => ROM_3
		EN --- EQ(ROM_SHU, 4) => ROM_4
		EN --- EQ(ROM_SHU, 5) => ROM_5
		EN --- EQ(ROM_SHU, 6) => ROM_6
		EN --- EQ(ROM_SHU, 7) => ROM_7
		EN --- EQ(ROM_SHU, 8) => ROM_8
		EN --- EQ(ROM_SHU, 9) => ROM_9
		EN --- EQ(ROM_SHU, 10) => ROM_10
		EN --- EQ(ROM_SHU, 11) => ROM_11
		EN --- EQ(ROM_SHU, 12) => ROM_12
		EN --- EQ(ROM_SHU, 13) => ROM_13
		EN --- EQ(ROM_SHU, 14) => ROM_14
		EN --- EQ(ROM_SHU, 0) => ROM_0
NETWORK 2
	*
		EN --- SEL(ROM_0, KU_SHU, 15) => KAIKU_SHU
NETWORK 3
	*
		EN --- SEL(ROM_1, SEL(ROM_2, SEL(ROM_3, SEL(ROM_4, SEL(ROM_5, SEL(ROM_6, SEL(ROM_7, SEL(ROM_8, SEL(ROM_9, SEL(ROM_10, SEL(ROM_11, SEL(ROM_12, SEL(ROM_13, SEL(ROM_14, 1, 1), 2), 3), 4), 5), 6), 7), 8), 9), 10), 11), 12), 13), 14) => KU_SHU
NETWORK 4
	*
		EN --- EQ(A_ROM, 15) => A_15
		EN --- EQ(A_ROM, 0) => A_0
		EN --- GE(A_ROM, KAIKU_SHU) => A_FJ
NETWORK 5
	[A_IN]
		EN --- MOVE(1) => ROM
NETWORK 6
	[A_FJ] - [CV_0]
		EN --- MOVE(1) => FJ_ROM
NETWORK 7
	[A_IN] - [A_0] --- (A_DZ)
NETWORK 8
	[INPUT_KA] - [A_FJ] - [/A_0] --- (A_KA)
NETWORK 9
	*
		EN --- EQ(B_ROM, 15) => B_15
		EN --- EQ(B_ROM, 0) => B_0
		EN --- GE(B_ROM, KAIKU_SHU) => B_FJ
NETWORK 10
	[B_IN]
		EN --- MOVE(2) => ROM
NETWORK 11
	[B_FJ] - [CV_1]
		EN --- MOVE(2) => FJ_ROM
NETWORK 12
	[B_IN] - [B_0] --- (B_DZ)
NETWORK 13
	[INPUT_KA] - [B_FJ] - [/B_0] --- (B_KA)
NETWORK 14
	*
		EN --- EQ(C_ROM, 15) => C_15
		EN --- EQ(C_ROM, 0) => C_0
		EN --- GE(C_ROM, KAIKU_SHU) => C_FJ
NETWORK 15
	[C_IN]
		EN --- MOVE(3) => ROM
NETWORK 16
	[C_FJ] - [CV_2]
		EN --- MOVE(3) => FJ_ROM
NETWORK 17
	[C_IN] - [C_0] --- (C_DZ)
NETWORK 18
	[INPUT_KA] - [C_FJ] - [/C_0] --- (C_KA)
NETWORK 19
	*
		EN --- EQ(D_ROM, 15) => D_15
		EN --- EQ(D_ROM, 0) => D_0
		EN --- GE(D_ROM, KAIKU_SHU) => D_FJ
NETWORK 20
	[D_IN]
		EN --- MOVE(4) => ROM
NETWORK 21
	[D_FJ] - [CV_3]
		EN --- MOVE(4) => FJ_ROM
NETWORK 22
	[D_IN] - [D_0] --- (D_DZ)
NETWORK 23
	[INPUT_KA] - [D_FJ] - [/D_0] --- (D_KA)
NETWORK 24
	*
		EN --- EQ(E_ROM, 15) => E_15
		EN --- EQ(E_ROM, 0) => E_0
		EN --- GE(E_ROM, KAIKU_SHU) => E_FJ
NETWORK 25
	[E_IN]
		EN --- MOVE(5) => ROM
NETWORK 26
	[E_FJ] - [CV_4]
		EN --- MOVE(5) => FJ_ROM
NETWORK 27
	[E_IN] - [E_0] --- (E_DZ)
NETWORK 28
	[INPUT_KA] - [E_FJ] - [/E_0] --- (E_KA)
NETWORK 29
	*
		EN --- EQ(F_ROM, 15) => F_15
		EN --- EQ(F_ROM, 0) => F_0
		EN --- GE(F_ROM, KAIKU_SHU) => F_FJ
NETWORK 30
	[F_IN]
		EN --- MOVE(6) => ROM
NETWORK 31
	[F_FJ] - [CV_5]
		EN --- MOVE(6) => FJ_ROM
NETWORK 32
	[F_IN] - [F_0] --- (F_DZ)
NETWORK 33
	[INPUT_KA] - [F_FJ] - [/F_0] --- (F_KA)
NETWORK 34
	*
		EN --- EQ(G_ROM, 15) => G_15
		EN --- EQ(G_ROM, 0) => G_0
		EN --- GE(G_ROM, KAIKU_SHU) => G_FJ
NETWORK 35
	[G_IN]
		EN --- MOVE(7) => ROM
NETWORK 36
	[G_FJ] - [CV_6]
		EN --- MOVE(7) => FJ_ROM
NETWORK 37
	[G_IN] - [G_0] --- (G_DZ)
NETWORK 38
	[INPUT_KA] - [G_FJ] - [/G_0] --- (G_KA)
NETWORK 39
	*
		EN --- EQ(H_ROM, 15) => H_15
		EN --- EQ(H_ROM, 0) => H_0
		EN --- GE(H_ROM, KAIKU_SHU) => H_FJ
NETWORK 40
	[H_IN]
		EN --- MOVE(8) => ROM
NETWORK 41
	[H_FJ] - [CV_7]
		EN --- MOVE(8) => FJ_ROM
NETWORK 42
	[H_IN] - [H_0] --- (H_DZ)
NETWORK 43
	[INPUT_KA] - [H_FJ] - [/H_0] --- (H_KA)
NETWORK 44
	*
		EN --- EQ(I_ROM, 15) => I_15
		EN --- EQ(I_ROM, 0) => I_0
		EN --- GE(I_ROM, KAIKU_SHU) => I_FJ
NETWORK 45
	[I_IN]
		EN --- MOVE(9) => ROM
NETWORK 46
	[I_FJ] - [CV_8]
		EN --- MOVE(9) => FJ_ROM
NETWORK 47
	[I_IN] - [I_0] --- (I_DZ)
NETWORK 48
	[INPUT_KA] - [I_FJ] - [/I_0] --- (I_KA)
NETWORK 49
	*
		EN --- EQ(J_ROM, 15) => J_15
		EN --- EQ(J_ROM, 0) => J_0
		EN --- GE(J_ROM, KAIKU_SHU) => J_FJ
NETWORK 50
	[J_IN]
		EN --- MOVE(10) => ROM
NETWORK 51
	[J_FJ] - [CV_9]
		EN --- MOVE(10) => FJ_ROM
NETWORK 52
	[J_IN] - [J_0] --- (J_DZ)
NETWORK 53
	[INPUT_KA] - [J_FJ] - [/J_0] --- (J_KA)
NETWORK 54
	*
		EN --- EQ(K_ROM, 15) => K_15
		EN --- EQ(K_ROM, 0) => K_0
		EN --- GE(K_ROM, KAIKU_SHU) => K_FJ
NETWORK 55
	[K_IN]
		EN --- MOVE(14) => ROM
NETWORK 56
	[K_FJ] - [CV_10]
		EN --- MOVE(14) => FJ_ROM
NETWORK 57
	[K_IN] - [K_0] --- (K_DZ)
NETWORK 58
	[INPUT_KA] - [K_FJ] - [/K_0] --- (K_KA)
NETWORK 59
	*
		EN --- EQ(L_ROM, 15) => L_15
		EN --- EQ(L_ROM, 0) => L_0
		EN --- GE(L_ROM, KAIKU_SHU) => L_FJ
NETWORK 60
	[L_IN]
		EN --- MOVE(11) => ROM
NETWORK 61
	[L_FJ] - [CV_11]
		EN --- MOVE(11) => FJ_ROM
NETWORK 62
	[L_IN] - [L_0] --- (L_DZ)
NETWORK 63
	[INPUT_KA] - [L_FJ] - [/L_0] --- (L_KA)
NETWORK 64
	*
		EN --- EQ(M_ROM, 15) => M_15
		EN --- EQ(M_ROM, 0) => M_0
		EN --- GE(M_ROM, KAIKU_SHU) => M_FJ
NETWORK 65
	[M_IN]
		EN --- MOVE(12) => ROM
NETWORK 66
	[M_FJ] - [CV_12]
		EN --- MOVE(12) => FJ_ROM
NETWORK 67
	[M_IN] - [M_0] --- (M_DZ)
NETWORK 68
	[INPUT_KA] - [M_FJ] - [/M_0] --- (M_KA)
NETWORK 69
	*
		EN --- EQ(N_ROM, 15) => N_15
		EN --- EQ(N_ROM, 0) => N_0
		EN --- GE(N_ROM, KAIKU_SHU) => N_FJ
NETWORK 70
	[N_IN]
		EN --- MOVE(13) => ROM
NETWORK 71
	[N_FJ] - [CV_13]
		EN --- MOVE(13) => FJ_ROM
NETWORK 72
	[N_IN] - [N_0] --- (N_DZ)
NETWORK 73
	[INPUT_KA] - [N_FJ] - [/N_0] --- (N_KA)
NETWORK 74
	*
		EN --- OR(A_IN, B_IN, C_IN, D_IN, E_IN, F_IN, G_IN, H_IN, I_IN, J_IN, K_IN, L_IN, M_IN, N_IN) => INPUT_KA
NETWORK 75
	[/INPUT_KA]
		EN --- MOVE(0) => ROM
NETWORK 76
	*
		EN --- OR(A_FJ, B_FJ, C_FJ, D_FJ, E_FJ, F_FJ, G_FJ, H_FJ, I_FJ, J_FJ, K_FJ, L_FJ, M_FJ, N_FJ) => KA_FJ
NETWORK 77
	[/KA_FJ]
		EN --- MOVE(0) => FJ_ROM
NETWORK 78
	[PSH_IN] - FJ_CTU:CTU(CU: *, RESET: CTU_Q, PV: 14, CV => CV) --- (CTU_Q)
NETWORK 79
	*
		EN --- EQ(0, CV) => CV_0
		EN --- EQ(1, CV) => CV_1
		EN --- EQ(2, CV) => CV_2
		EN --- EQ(3, CV) => CV_3
		EN --- EQ(4, CV) => CV_4
		EN --- EQ(5, CV) => CV_5
		EN --- EQ(6, CV) => CV_6
		EN --- EQ(7, CV) => CV_7
		EN --- EQ(8, CV) => CV_8
		EN --- EQ(9, CV) => CV_9
		EN --- EQ(10, CV) => CV_10
		EN --- EQ(11, CV) => CV_11
		EN --- EQ(12, CV) => CV_12
		EN --- EQ(13, CV) => CV_13
_END_LD_
(* the same logic as Structured Text *)
(* Network 1 *)
ROM_1 := ROM_SHU = 1;
ROM_2 := ROM_SHU = 2;
ROM_3 := ROM_SHU = 3;
ROM_4 := ROM_SHU = 4;
ROM_5 := ROM_SHU = 5;
ROM_6 := ROM_SHU = 6;
ROM_7 := ROM_SHU = 7;
ROM_8 := ROM_SHU = 8;
ROM_9 := ROM_SHU = 9;
ROM_10 := ROM_SHU = 10;
ROM_11 := ROM_SHU = 11;
ROM_12 := ROM_SHU = 12;
ROM_13 := ROM_SHU = 13;
ROM_14 := ROM_SHU = 14;
ROM_0 := ROM_SHU = 0;
(* Network 2 *)
KAIKU_SHU := SEL(ROM_0, KU_SHU, 15);
(* Network 3 *)
KU_SHU := SEL(ROM_1, SEL(ROM_2, SEL(ROM_3, SEL(ROM_4, SEL(ROM_5, SEL(ROM_6, SEL(ROM_7, SEL(ROM_8, SEL(ROM_9, SEL(ROM_10, SEL(ROM_11, SEL(ROM_12, SEL(ROM_13, SEL(ROM_14, 1, 1), 2), 3), 4), 5), 6), 7), 8), 9), 10), 11), 12), 13), 14);
(* Network 4 *)
A_15 := A_ROM = 15;
A_0 := A_ROM = 0;
A_FJ := A_ROM >= KAIKU_SHU;
(* Network 5 *)
IF A_IN THEN
	ROM := 1;
END_IF;
(* Network 6 *)
IF A_FJ AND CV_0 THEN
	FJ_ROM := 1;
END_IF;
(* Network 7 *)
A_DZ := A_IN AND A_0;
(* Network 8 *)
A_KA := INPUT_KA AND A_FJ AND NOT A_0;
(* Network 9 *)
B_15 := B_ROM = 15;
B_0 := B_ROM = 0;
B_FJ := B_ROM >= KAIKU_SHU;
(* Network 10 *)
IF B_IN THEN
	ROM := 2;
END_IF;
(* Network 11 *)
IF B_FJ AND CV_1 THEN
	FJ_ROM := 2;
END_IF;
(* Network 12 *)
B_DZ := B_IN AND B_0;
(* Network 13 *)
B_KA := INPUT_KA AND B_FJ AND NOT B_0;
(* Network 14 *)
C_15 := C_ROM = 15;
C_0 := C_ROM = 0;
C_FJ := C_ROM >= KAIKU_SHU;
(* Network 15 *)
IF C_IN THEN
	ROM := 3;
END_IF;
(* Network 16 *)
IF C_FJ AND CV_2 THEN
	FJ_ROM := 3;
END_IF;
(* Network 17 *)
C_DZ := C_IN AND C_0;
(* Network 18 *)
C_KA := INPUT_KA AND C_FJ AND NOT C_0;
(* Network 19 *)
D_15 := D_ROM = 15;
D_0 := D_ROM = 0;
D_FJ := D_ROM >= KAIKU_SHU;
(* Network 20 *)
IF D_IN THEN
	ROM := 4;
END_IF;
(* Network 21 *)
IF D_FJ AND CV_3 THEN
	FJ_ROM := 4;
END_IF;
(* Network 22 *)
D_DZ := D_IN AND D_0;
(* Network 23 *)
D_KA := INPUT_KA AND D_FJ AND NOT D_0;
(* Network 24 *)
E_15 := E_ROM = 15;
E_0 := E_ROM = 0;
E_FJ := E_ROM >= KAIKU_SHU;
(* Network 25 *)
IF E_IN THEN
	ROM := 5;
END_IF;
(* Network 26 *)
IF E_FJ AND CV_4 THEN
	FJ_ROM := 5;
END_IF;
(* Network 27 *)
E_DZ := E_IN AND E_0;
(* Network 28 *)
E_KA := INPUT_KA AND E_FJ AND NOT E_0;
(* Network 29 *)
F_15 := F_ROM = 15;
F_0 := F_ROM = 0;
F_FJ := F_ROM >= KAIKU_SHU;
(* Network 30 *)
IF F_IN THEN
	ROM := 6;
END_IF;
(* Network 31 *)
IF F_FJ AND CV_5 THEN
	FJ_ROM := 6;
END_IF;
(* Network 32 *)
F_DZ := F_IN AND F_0;
(* Network 33 *)
F_KA := INPUT_KA AND F_FJ AND NOT F_0;
(* Network 34 *)
G_15 := G_ROM = 15;
G_0 := G_ROM = 0;
G_FJ := G_ROM >= KAIKU_SHU;
(* Network 35 *)
IF G_IN THEN
	ROM := 7;
END_IF;
(* Network 36 *)
IF G_FJ AND CV_6 THEN
	FJ_ROM := 7;
END_IF;
(* Network 37 *)
G_DZ := G_IN AND G_0;
(* Network 38 *)
G_KA := INPUT_KA AND G_FJ AND NOT G_0;
(* Network 39 *)
H_15 := H_ROM = 15;
H_0 := H_ROM = 0;
H_FJ := H_ROM >= KAIKU_SHU;
(* Network 40 *)
IF H_IN THEN
	ROM := 8;
END_IF;
(* Network 41 *)
IF H_FJ AND CV_7 THEN
	FJ_ROM := 8;
END_IF;
(* Network 42 *)
H_DZ := H_IN AND H_0;
(* Network 43 *)
H_KA := INPUT_KA AND H_FJ AND NOT H_0;
(* Network 44 *)
I_15 := I_ROM = 15;
I_0 := I_ROM = 0;
I_FJ := I_ROM >= KAIKU_SHU;
(* Network 45 *)
IF I_IN THEN
	ROM := 9;
END_IF;
(* Network 46 *)
IF I_FJ AND CV_8 THEN
	FJ_ROM := 9;
END_IF;
(* Network 47 *)
I_DZ := I_IN AND I_0;
(* Network 48 *)
I_KA := INPUT_KA AND I_FJ AND NOT I_0;
(* Network 49 *)
J_15 := J_ROM = 15;
J_0 := J_ROM = 0;
J_FJ := J_ROM >= KAIKU_SHU;
(* Network 50 *)
IF J_IN THEN
	ROM := 10;
END_IF;
(* Network 51 *)
IF J_FJ AND CV_9 THEN
	FJ_ROM := 10;
END_IF;
(* Network 52 *)
J_DZ := J_IN AND J_0;
(* Network 53 *)
J_KA := INPUT_KA AND J_FJ AND NOT J_0;
(* Network 54 *)
K_15 := K_ROM = 15;
K_0 := K_ROM = 0;
K_FJ := K_ROM >= KAIKU_SHU;
(* Network 55 *)
IF K_IN THEN
	ROM := 14;
END_IF;
(* Network 56 *)
IF K_FJ AND CV_10 THEN
	FJ_ROM := 14;
END_IF;
(* Network 57 *)
K_DZ := K_IN AND K_0;
(* Network 58 *)
K_KA := INPUT_KA AND K_FJ AND NOT K_0;
(* Network 59 *)
L_15 := L_ROM = 15;
L_0 := L_ROM = 0;
L_FJ := L_ROM >= KAIKU_SHU;
(* Network 60 *)
IF L_IN THEN
	ROM := 11;
END_IF;
(* Network 61 *)
IF L_FJ AND CV_11 THEN
	FJ_ROM := 11;
END_IF;
(* Network 62 *)
L_DZ := L_IN AND L_0;
(* Network 63 *)
L_KA := INPUT_KA AND L_FJ AND NOT L_0;
(* Network 64 *)
M_15 := M_ROM = 15;
M_0 := M_ROM = 0;
M_FJ := M_ROM >= KAIKU_SHU;
(* Network 65 *)
IF M_IN THEN
	ROM := 12;
END_IF;
(* Network 66 *)
IF M_FJ AND CV_12 THEN
	FJ_ROM := 12;
END_IF;
(* Network 67 *)
M_DZ := M_IN AND M_0;
(* Network 68 *)
M_KA := INPUT_KA AND M_FJ AND NOT M_0;
(* Network 69 *)
N_15 := N_ROM = 15;
N_0 := N_ROM = 0;
N_FJ := N_ROM >= KAIKU_SHU;
(* Network 70 *)
IF N_IN THEN
	ROM := 13;
END_IF;
(* Network 71 *)
IF N_FJ AND CV_13 THEN
	FJ_ROM := 13;
END_IF;
(* Network 72 *)
N_DZ := N_IN AND N_0;
(* Network 73 *)
N_KA := INPUT_KA AND N_FJ AND NOT N_0;
(* Network 74 *)
INPUT_KA := A_IN OR B_IN OR C_IN OR D_IN OR E_IN OR F_IN OR G_IN OR H_IN OR I_IN OR J_IN OR K_IN OR L_IN OR M_IN OR N_IN;
(* Network 75 *)
IF NOT INPUT_KA THEN
	ROM := 0;
END_IF;
(* Network 76 *)
KA_FJ := A_FJ OR B_FJ OR C_FJ OR D_FJ OR E_FJ OR F_FJ OR G_FJ OR H_FJ OR I_FJ OR J_FJ OR K_FJ OR L_FJ OR M_FJ OR N_FJ;
(* Network 77 *)
IF NOT KA_FJ THEN
	FJ_ROM := 0;
END_IF;
(* Network 78 *)
FJ_CTU(CU := PSH_IN, RESET := CTU_Q, PV := 14);
CV := FJ_CTU.CV;
CTU_Q := FJ_CTU.Q;
(* Network 79 *)
CV_0 := 0 = CV;
CV_1 := 1 = CV;
CV_2 := 2 = CV;
CV_3 := 3 = CV;
CV_4 := 4 = CV;
CV_5 := 5 = CV;
CV_6 := 6 = CV;
CV_7 := 7 = CV;
CV_8 := 8 = CV;
CV_9 := 9 = CV;
CV_10 := 10 = CV;
CV_11 := 11 = CV;
CV_12 := 12 = CV;
CV_13 := 13 = CV;
END_FUNCTION_BLOCK

(* POU PQ_GRD, LD *)
FUNCTION_BLOCK PQ_GRD
VAR_INPUT
	PQ_YA_IN: INT;
	PQ_WD_IN: INT;
	PQ_GRD_SET: INT;
	GRD_YSH_SET: WORD;
	OPEN_IN: BOOL;
	RESET: BOOL;
END_VAR
VAR_OUTPUT
	PQ_BH_WD: INT;
	PQ_GRD_OUT: INT;

	GRD_ALA: BOOL;
	GRD_YSH: WORD;
END_VAR
VAR
	YL_WD: YL_WD;
	GRD_KA: BOOL;
	GRD_YSH_EQ0: BOOL;
	YANSHI_OPEN: YANSHI_OPEN;
END_VAR
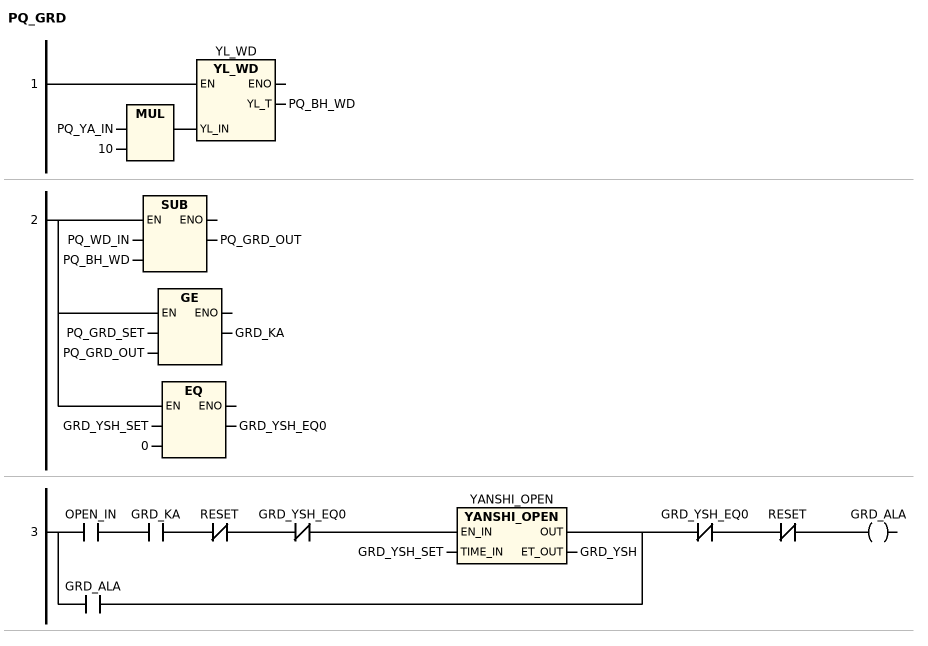
_LD_ (* Ladder Diagram *)
NETWORK 1
	*
		EN --- YL_WD:YL_WD(YL_IN: MUL(PQ_YA_IN, 10)) => PQ_BH_WD
NETWORK 2
	*
		EN --- SUB(PQ_WD_IN, PQ_BH_WD) => PQ_GRD_OUT
		EN --- GE(PQ_GRD_SET, PQ_GRD_OUT) => GRD_KA
		EN --- EQ(GRD_YSH_SET, 0) => GRD_YSH_EQ0
NETWORK 3
	{ [OPEN_IN] - [GRD_KA] - [/RESET] - [/GRD_YSH_EQ0] - YANSHI_OPEN:YANSHI_OPEN(EN_IN: *, TIME_IN: GRD_YSH_SET, ET_OUT => GRD_YSH) | [GRD_ALA] } - [/GRD_YSH_EQ0] - [/RESET] --- (GRD_ALA)
_END_LD_
(* the same logic as Structured Text *)
(* Network 1 *)
YL_WD(YL_IN := PQ_YA_IN * 10);
PQ_BH_WD := YL_WD.YL_T;
(* Network 2 *)
PQ_GRD_OUT := PQ_WD_IN - PQ_BH_WD;
GRD_KA := PQ_GRD_SET >= PQ_GRD_OUT;
GRD_YSH_EQ0 := GRD_YSH_SET = 0;
(* Network 3 *)
YANSHI_OPEN(EN_IN := OPEN_IN AND GRD_KA AND NOT RESET AND NOT GRD_YSH_EQ0, TIME_IN := GRD_YSH_SET);
GRD_YSH := YANSHI_OPEN.ET_OUT;
GRD_ALA := (YANSHI_OPEN.OUT OR GRD_ALA) AND NOT GRD_YSH_EQ0 AND NOT RESET;
END_FUNCTION_BLOCK

(* POU SHL_BH, LD *)
FUNCTION_BLOCK  SHL_BH
VAR
	SHL_Y: YANSHI_OPEN;
	SET_0: BOOL;
END_VAR
VAR_INPUT
	OPEN_IN: BOOL;
	SHL_IN: BOOL;
	SHL_YSH_SET: WORD;
	RESET: BOOL;
END_VAR
VAR_OUTPUT
	SHL_ALA: BOOL;
	SHB_KA: BOOL;
	SHL_YSH_XH: WORD;

	KJ_OUT: BOOL;
END_VAR
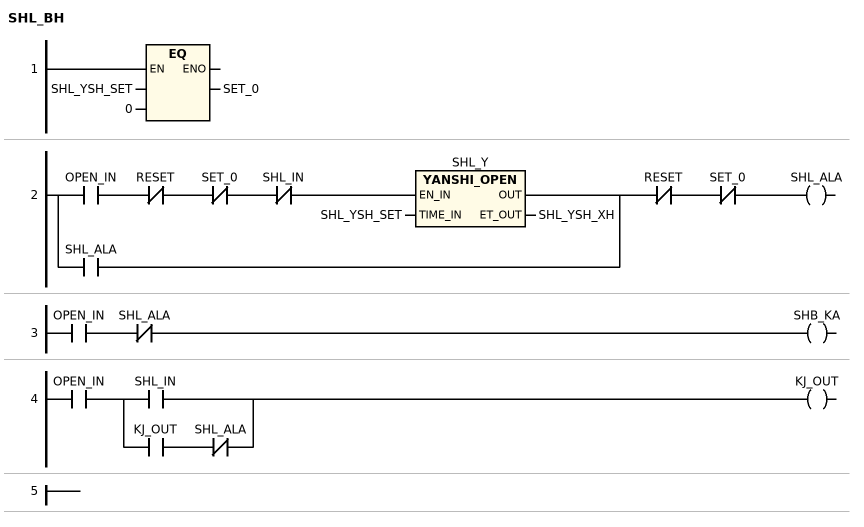
_LD_ (* Ladder Diagram *)
NETWORK 1
	*
		EN --- EQ(SHL_YSH_SET, 0) => SET_0
NETWORK 2
	{ [OPEN_IN] - [/RESET] - [/SET_0] - [/SHL_IN] - SHL_Y:YANSHI_OPEN(EN_IN: *, TIME_IN: SHL_YSH_SET, ET_OUT => SHL_YSH_XH) | [SHL_ALA] } - [/RESET] - [/SET_0] --- (SHL_ALA)
NETWORK 3
	[OPEN_IN] - [/SHL_ALA] --- (SHB_KA)
NETWORK 4
	[OPEN_IN] - { [SHL_IN] | [KJ_OUT] - [/SHL_ALA] } --- (KJ_OUT)
NETWORK 5
	*
_END_LD_
(* the same logic as Structured Text *)
(* Network 1 *)
SET_0 := SHL_YSH_SET = 0;
(* Network 2 *)
SHL_Y(EN_IN := OPEN_IN AND NOT RESET AND NOT SET_0 AND NOT SHL_IN, TIME_IN := SHL_YSH_SET);
SHL_YSH_XH := SHL_Y.ET_OUT;
SHL_ALA := (SHL_Y.OUT OR SHL_ALA) AND NOT RESET AND NOT SET_0;
(* Network 3 *)
SHB_KA := OPEN_IN AND NOT SHL_ALA;
(* Network 4 *)
KJ_OUT := OPEN_IN AND (SHL_IN OR KJ_OUT AND NOT SHL_ALA);
(* Network 5 *)
END_FUNCTION_BLOCK

(* POU BJ_MIN_COOL_1, LD *)
FUNCTION_BLOCK BJ_MIN_COOL_1
VAR_INPUT
	XH_SHU: WORD;
	ONE_H_IN: DWORD;
	TWO_H_IN: DWORD;
	THREE_H_IN: DWORD;
	FOUER_H_IN: DWORD;
	FIVE_H_IN: DWORD;
	SIX_H_IN: DWORD;
	CHD_ONE_IN: BOOL;
	CHD_TWO_IN: BOOL;
	CHD_THREE_IN: BOOL;
	CHD_FOUER_IN: BOOL;
	CHD_FIVE_IN: BOOL;
	CHD_SIX_IN: BOOL;
	FW_1: BOOL;
	FW_2: BOOL;
	FW_3: BOOL;
	FW_4: BOOL;
	FW_5: BOOL;
	FW_6: BOOL;
END_VAR
VAR_OUTPUT
	ONE_CX_1: BYTE;
	TWO_CX_1: BYTE;
	THREE_CX_1: BYTE;
	FOUER_CX_1: BYTE;
	FIVE_CX_1: BYTE;
	SIX_CX_1: BYTE;
	ONE_CIXU: BYTE;
	TWO_CIXU: BYTE;
	THREE_CIXU: BYTE;
	FOUER_CIXU: BYTE;
	FIVE_CIXU: BYTE;
	SIX_CIXU: BYTE;
END_VAR
VAR
	ONE_H_ZC_1: DWORD;
	TWO_H_ZC_1: DWORD;
	THREE_H_ZC_1: DWORD;
	FOUER_H_ZC_1: DWORD;
	FIVE_H_ZC_1: DWORD;
	ONE_CX_ZC: BYTE;
	TWO_CX_ZC: BYTE;
	THREE_CX_ZC: BYTE;
	FOUER_CX_ZC: BYTE;
	FIVE_CX_ZC: BYTE;
	ONE_H_ZC_2: DWORD;
	TWO_H_ZC_2: DWORD;
	THREE_H_ZC_2: DWORD;
	FOUER_H_ZC_2: DWORD;
	FIVE_H_ZC_2: DWORD;
	ONE_FUWEI: BOOL;
	TWO_FUWEI: BOOL;
	FIVE_FUWEI: BOOL;
	FOUER_FUWEI: BOOL;
	THREE_FUWEI: BOOL;
	R1_IN: R_TRIG;
	BJ_COOL: BJ_CIXU_COOL;
	SIX_H_ZC_1: DWORD;
	SIX_CX_ZC: BYTE;
	SIX_FUWEI: BOOL;
	SIX_H_ZC_2: DWORD;
	OPEN_KA: BOOL;

	TWO_CX_2: BYTE;

	BJ_CX: BJ_CIXU_COOL;
	FW_CX_6: BOOL;
	FW_CX_5: BOOL;
	FW_CX_4: BOOL;
	FW_CX_3: BOOL;
	FW_CX_2: BOOL;
	FW_CX_1: BOOL;
	JQ1_CX_6: BOOL;
	JQ1_CX_1: BOOL;
	JQ1_CX_2: BOOL;
	JQ1_CX_3: BOOL;
	JQ_CX_1: BOOL;
	JQ1_CX_KG_1: BOOL;
	JQ1_CX_KG_2: BOOL;
	JQ1_CX_KG_3: BOOL;
	JQ1_CX_KG_4: BOOL;
	JQ1_CX_KG_5: BOOL;
	JQ1_CX_KG_6: BOOL;
	JQ2_CX_KG_1: BOOL;
	JQ2_CX_KG_2: BOOL;
	JQ2_CX_KG_3: BOOL;
	JQ2_CX_KG_4: BOOL;
	JQ2_CX_KG_5: BOOL;
	JQ2_CX_KG_6: BOOL;
	JQ3_CX_KG_1: BOOL;
	JQ3_CX_KG_2: BOOL;
	JQ3_CX_KG_3: BOOL;
	JQ3_CX_KG_4: BOOL;
	JQ3_CX_KG_5: BOOL;
	JQ3_CX_KG_6: BOOL;
	JQ4_CX_KG_1: BOOL;
	JQ4_CX_KG_2: BOOL;
	JQ4_CX_KG_3: BOOL;
	JQ4_CX_KG_4: BOOL;
	JQ4_CX_KG_5: BOOL;
	JQ4_CX_KG_6: BOOL;
	JQ5_CX_KG_1: BOOL;
	JQ5_CX_KG_2: BOOL;
	JQ5_CX_KG_3: BOOL;
	JQ5_CX_KG_4: BOOL;
	JQ5_CX_KG_5: BOOL;
	JQ5_CX_KG_6: BOOL;
	JQ6_CX_KG_1: BOOL;
	JQ6_CX_KG_2: BOOL;
	JQ6_CX_KG_3: BOOL;
	JQ6_CX_KG_4: BOOL;
	JQ6_CX_KG_5: BOOL;
	JQ6_CX_KG_6: BOOL;
	JQ_1_FW: BOOL;
END_VAR
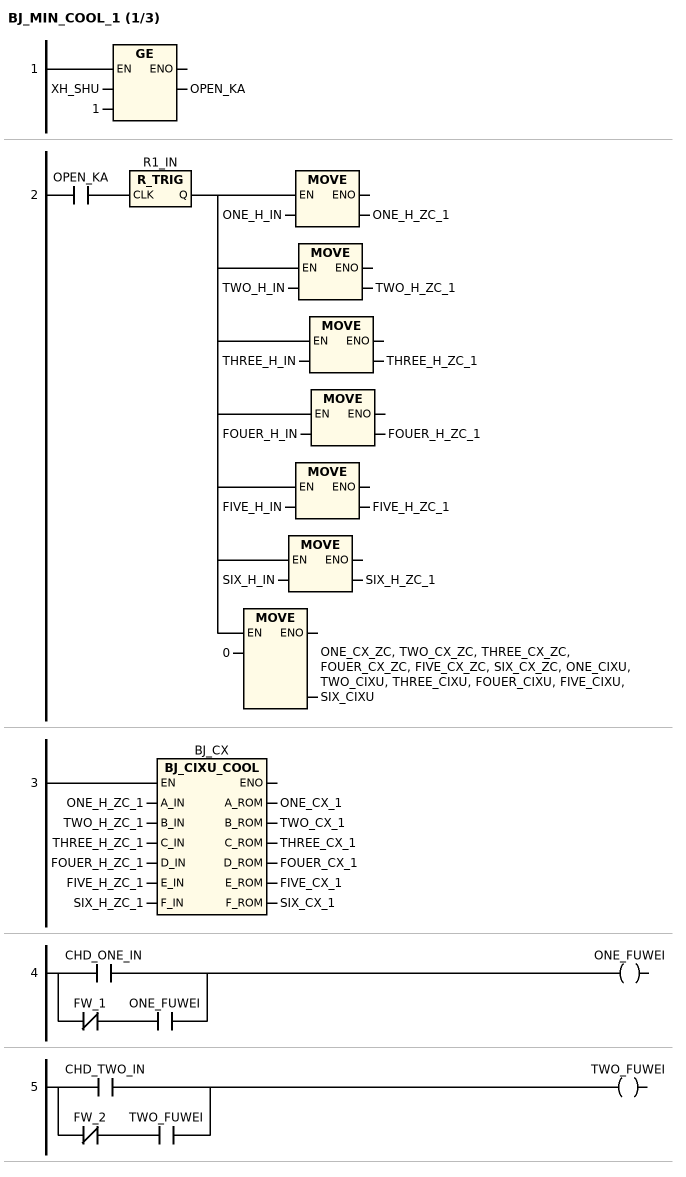
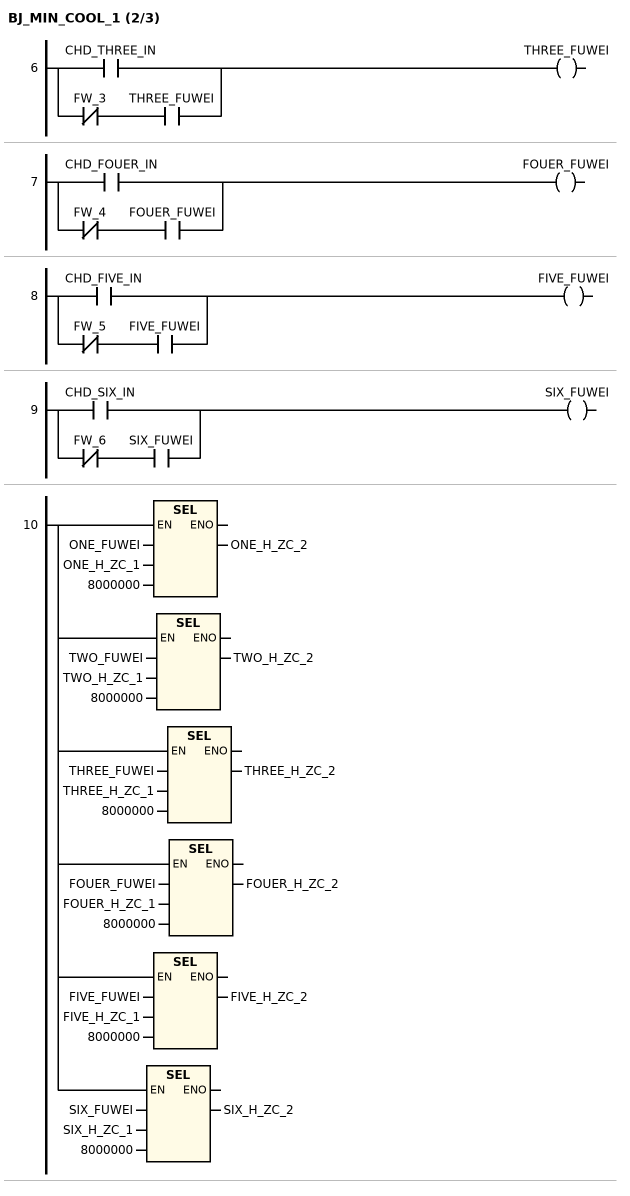
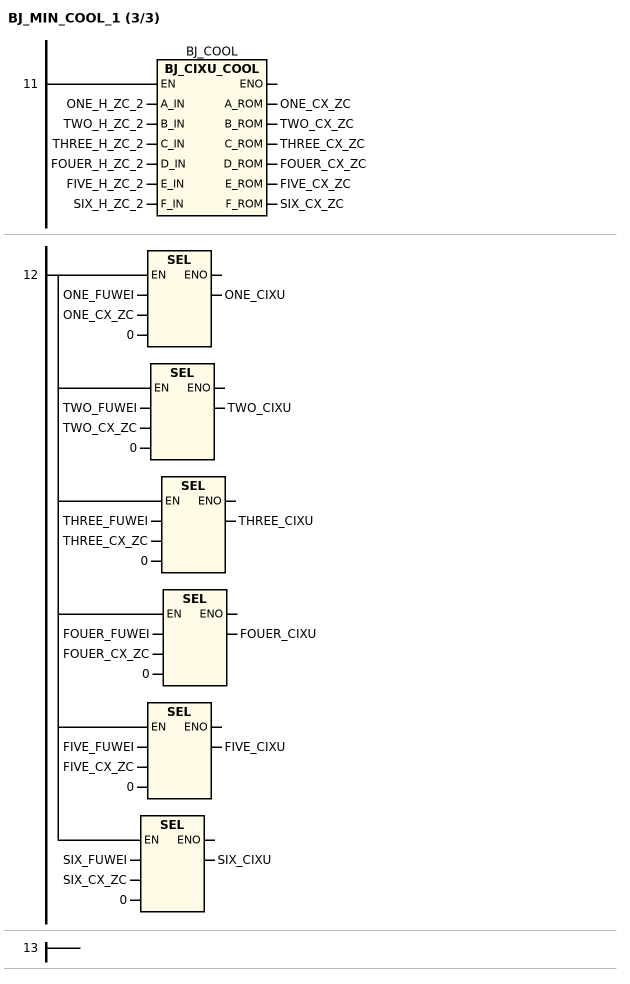
_LD_ (* Ladder Diagram *)
NETWORK 1
	*
		EN --- GE(XH_SHU, 1) => OPEN_KA
NETWORK 2
	[OPEN_KA] - R1_IN:R_TRIG(CLK: *)
		EN --- MOVE(ONE_H_IN) => ONE_H_ZC_1
		EN --- MOVE(TWO_H_IN) => TWO_H_ZC_1
		EN --- MOVE(THREE_H_IN) => THREE_H_ZC_1
		EN --- MOVE(FOUER_H_IN) => FOUER_H_ZC_1
		EN --- MOVE(FIVE_H_IN) => FIVE_H_ZC_1
		EN --- MOVE(SIX_H_IN) => SIX_H_ZC_1
		EN --- MOVE(0) => ONE_CX_ZC, TWO_CX_ZC, THREE_CX_ZC, FOUER_CX_ZC, FIVE_CX_ZC, SIX_CX_ZC, ONE_CIXU, TWO_CIXU, THREE_CIXU, FOUER_CIXU, FIVE_CIXU, SIX_CIXU
NETWORK 3
	*
		EN --- BJ_CX:BJ_CIXU_COOL(A_IN: ONE_H_ZC_1, B_IN: TWO_H_ZC_1, C_IN: THREE_H_ZC_1, D_IN: FOUER_H_ZC_1, E_IN: FIVE_H_ZC_1, F_IN: SIX_H_ZC_1, B_ROM => TWO_CX_1, C_ROM => THREE_CX_1, D_ROM => FOUER_CX_1, E_ROM => FIVE_CX_1, F_ROM => SIX_CX_1) => ONE_CX_1
NETWORK 4
	{ [CHD_ONE_IN] | [/FW_1] - [ONE_FUWEI] } --- (ONE_FUWEI)
NETWORK 5
	{ [CHD_TWO_IN] | [/FW_2] - [TWO_FUWEI] } --- (TWO_FUWEI)
NETWORK 6
	{ [CHD_THREE_IN] | [/FW_3] - [THREE_FUWEI] } --- (THREE_FUWEI)
NETWORK 7
	{ [CHD_FOUER_IN] | [/FW_4] - [FOUER_FUWEI] } --- (FOUER_FUWEI)
NETWORK 8
	{ [CHD_FIVE_IN] | [/FW_5] - [FIVE_FUWEI] } --- (FIVE_FUWEI)
NETWORK 9
	{ [CHD_SIX_IN] | [/FW_6] - [SIX_FUWEI] } --- (SIX_FUWEI)
NETWORK 10
	*
		EN --- SEL(ONE_FUWEI, ONE_H_ZC_1, 8000000) => ONE_H_ZC_2
		EN --- SEL(TWO_FUWEI, TWO_H_ZC_1, 8000000) => TWO_H_ZC_2
		EN --- SEL(THREE_FUWEI, THREE_H_ZC_1, 8000000) => THREE_H_ZC_2
		EN --- SEL(FOUER_FUWEI, FOUER_H_ZC_1, 8000000) => FOUER_H_ZC_2
		EN --- SEL(FIVE_FUWEI, FIVE_H_ZC_1, 8000000) => FIVE_H_ZC_2
		EN --- SEL(SIX_FUWEI, SIX_H_ZC_1, 8000000) => SIX_H_ZC_2
NETWORK 11
	*
		EN --- BJ_COOL:BJ_CIXU_COOL(A_IN: ONE_H_ZC_2, B_IN: TWO_H_ZC_2, C_IN: THREE_H_ZC_2, D_IN: FOUER_H_ZC_2, E_IN: FIVE_H_ZC_2, F_IN: SIX_H_ZC_2, B_ROM => TWO_CX_ZC, C_ROM => THREE_CX_ZC, D_ROM => FOUER_CX_ZC, E_ROM => FIVE_CX_ZC, F_ROM => SIX_CX_ZC) => ONE_CX_ZC
NETWORK 12
	*
		EN --- SEL(ONE_FUWEI, ONE_CX_ZC, 0) => ONE_CIXU
		EN --- SEL(TWO_FUWEI, TWO_CX_ZC, 0) => TWO_CIXU
		EN --- SEL(THREE_FUWEI, THREE_CX_ZC, 0) => THREE_CIXU
		EN --- SEL(FOUER_FUWEI, FOUER_CX_ZC, 0) => FOUER_CIXU
		EN --- SEL(FIVE_FUWEI, FIVE_CX_ZC, 0) => FIVE_CIXU
		EN --- SEL(SIX_FUWEI, SIX_CX_ZC, 0) => SIX_CIXU
NETWORK 13
	*
_END_LD_
(* the same logic as Structured Text *)
(* Network 1 *)
OPEN_KA := XH_SHU >= 1;
(* Network 2: see the listing above *)
(* Network 3 *)
BJ_CX(A_IN := ONE_H_ZC_1, B_IN := TWO_H_ZC_1, C_IN := THREE_H_ZC_1, D_IN := FOUER_H_ZC_1, E_IN := FIVE_H_ZC_1, F_IN := SIX_H_ZC_1);
TWO_CX_1 := BJ_CX.B_ROM;
THREE_CX_1 := BJ_CX.C_ROM;
FOUER_CX_1 := BJ_CX.D_ROM;
FIVE_CX_1 := BJ_CX.E_ROM;
SIX_CX_1 := BJ_CX.F_ROM;
ONE_CX_1 := BJ_CX.A_ROM;
(* Network 4 *)
ONE_FUWEI := CHD_ONE_IN OR NOT FW_1 AND ONE_FUWEI;
(* Network 5 *)
TWO_FUWEI := CHD_TWO_IN OR NOT FW_2 AND TWO_FUWEI;
(* Network 6 *)
THREE_FUWEI := CHD_THREE_IN OR NOT FW_3 AND THREE_FUWEI;
(* Network 7 *)
FOUER_FUWEI := CHD_FOUER_IN OR NOT FW_4 AND FOUER_FUWEI;
(* Network 8 *)
FIVE_FUWEI := CHD_FIVE_IN OR NOT FW_5 AND FIVE_FUWEI;
(* Network 9 *)
SIX_FUWEI := CHD_SIX_IN OR NOT FW_6 AND SIX_FUWEI;
(* Network 10 *)
ONE_H_ZC_2 := SEL(ONE_FUWEI, ONE_H_ZC_1, 8000000);
TWO_H_ZC_2 := SEL(TWO_FUWEI, TWO_H_ZC_1, 8000000);
THREE_H_ZC_2 := SEL(THREE_FUWEI, THREE_H_ZC_1, 8000000);
FOUER_H_ZC_2 := SEL(FOUER_FUWEI, FOUER_H_ZC_1, 8000000);
FIVE_H_ZC_2 := SEL(FIVE_FUWEI, FIVE_H_ZC_1, 8000000);
SIX_H_ZC_2 := SEL(SIX_FUWEI, SIX_H_ZC_1, 8000000);
(* Network 11 *)
BJ_COOL(A_IN := ONE_H_ZC_2, B_IN := TWO_H_ZC_2, C_IN := THREE_H_ZC_2, D_IN := FOUER_H_ZC_2, E_IN := FIVE_H_ZC_2, F_IN := SIX_H_ZC_2);
TWO_CX_ZC := BJ_COOL.B_ROM;
THREE_CX_ZC := BJ_COOL.C_ROM;
FOUER_CX_ZC := BJ_COOL.D_ROM;
FIVE_CX_ZC := BJ_COOL.E_ROM;
SIX_CX_ZC := BJ_COOL.F_ROM;
ONE_CX_ZC := BJ_COOL.A_ROM;
(* Network 12 *)
ONE_CIXU := SEL(ONE_FUWEI, ONE_CX_ZC, 0);
TWO_CIXU := SEL(TWO_FUWEI, TWO_CX_ZC, 0);
THREE_CIXU := SEL(THREE_FUWEI, THREE_CX_ZC, 0);
FOUER_CIXU := SEL(FOUER_FUWEI, FOUER_CX_ZC, 0);
FIVE_CIXU := SEL(FIVE_FUWEI, FIVE_CX_ZC, 0);
SIX_CIXU := SEL(SIX_FUWEI, SIX_CX_ZC, 0);
(* Network 13: see the listing above *)
END_FUNCTION_BLOCK

(* POU BJ_FUWEI_1, LD *)
FUNCTION_BLOCK BJ_FUWEI_1
VAR_INPUT
	XH_SHUI: WORD;
	JQ_1: BOOL;
	JQ_2: BOOL;
	JQ_3: BOOL;
	JQ_4: BOOL;
	JQ_5: BOOL;
	JQ_6: BOOL;
	CX_1: BYTE;
	CX_2: BYTE;
	CX_3: BYTE;
	CX_4: BYTE;
	CX_5: BYTE;
	CX_6: BYTE;
	CX_1_1: BYTE;
	CX_2_1: BYTE;
	CX_3_1: BYTE;
	CX_4_1: BYTE;
	CX_5_1: BYTE;
	CX_6_1: BYTE;
	CHD_1: BOOL;
	CHD_2: BOOL;
	CHD_3: BOOL;
	CHD_4: BOOL;
	CHD_5: BOOL;
	CHD_6: BOOL;
END_VAR
VAR_OUTPUT
	FW_1: BOOL;
	FW_2: BOOL;
	FW_3: BOOL;
	FW_4: BOOL;
	FW_5: BOOL;
	FW_6: BOOL;
	FS_KA: BOOL;
	JZ_OUT: BOOL;
END_VAR
VAR
	JT_A_SHU: WORD;
	JT_B_SHU: WORD;
	FUWEI_A_3: BOOL;
	FUWEI_B_3: BOOL;
	FUWEI_A_1: BOOL;
	FUWEI_B_1: BOOL;
	FUWEI_A_2: BOOL;
	FUWEI_B_2: BOOL;
	JQ_A_SHU: WORD;
	JQ_B_SHU: WORD;
	XH_SHU: WORD;
	JQ_SHU: WORD;
	CX_MAX: BYTE;
	CX_MAX_1: BOOL;
	CX_MAX_2: BOOL;
	CX_MAX_3: BOOL;
	CX_MAX_4: BOOL;
	CX_MAX_5: BOOL;
	CX_MAX_6: BOOL;
	FUWEI_1: BOOL;

	FW: BOOL;
	CX_MAX2: BYTE;
	CX_MAX2_1: BOOL;
	CX_MAX2_2: BOOL;
	CX_MAX2_3: BOOL;
	CX_MAX2_4: BOOL;
	CX_MAX2_5: BOOL;
	CX_MAX2_6: BOOL;
	CX_MAX1: BYTE;
	A: BOOL;
	B: BOOL;
	C: BOOL;

END_VAR
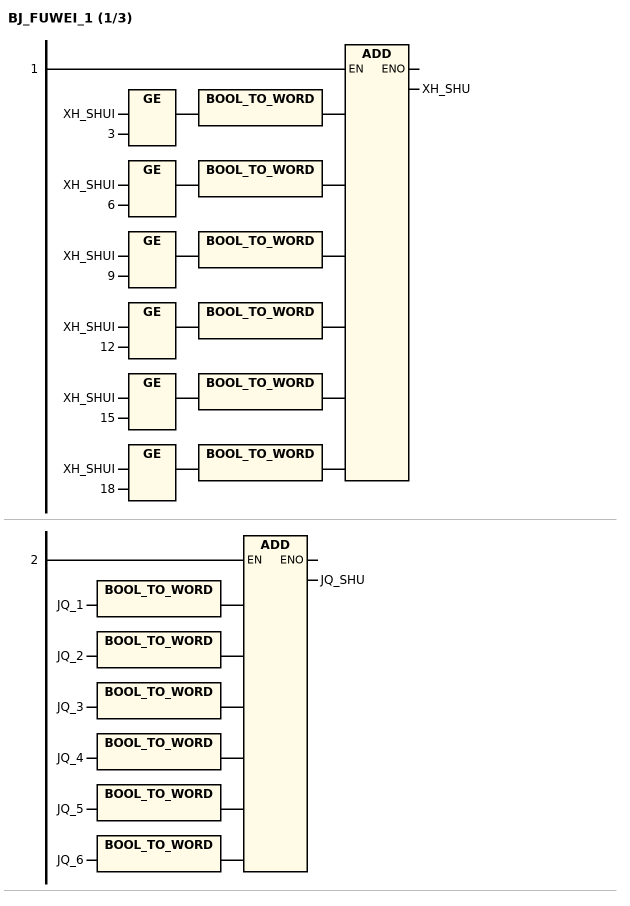
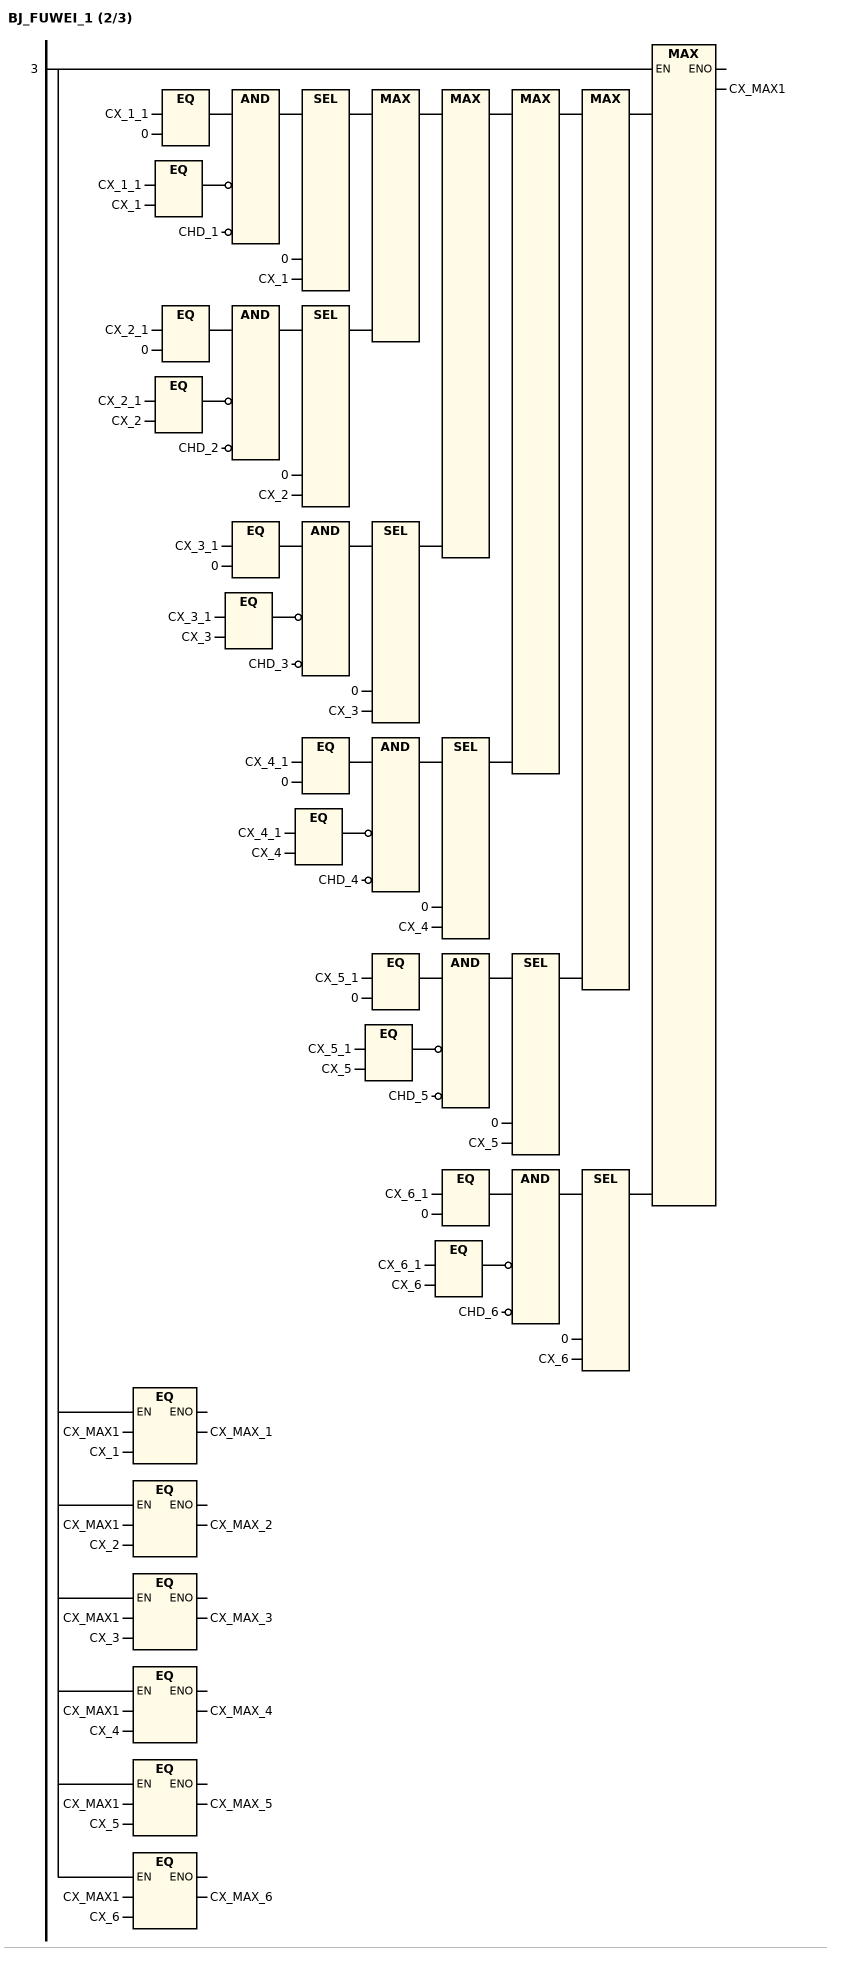
